KUKA KRL program: MyProgram_325().src

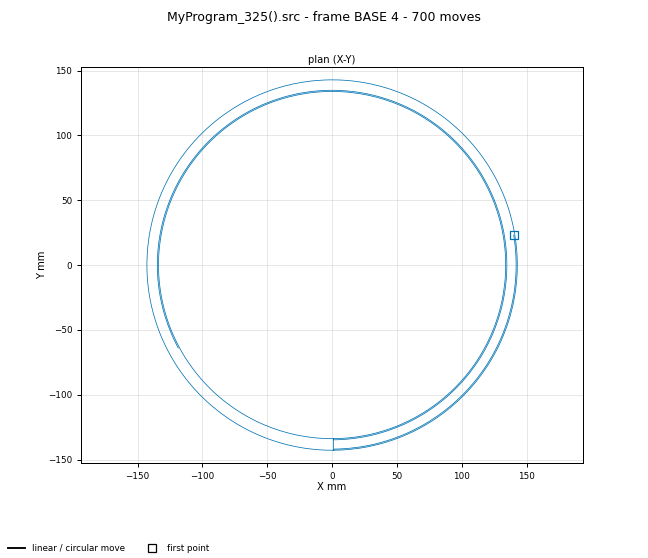
[picture p0: tool path of MyProgram_325().src in frame BASE 4, 700 of 700 moves have a stored position in this frame; points joined in program order, loops and branches not executed]
&ACCESS RVP
&REL 1
&PARAM TEMPLATE = C:\KRC\Roboter\Template\vorgabe
&PARAM EDITMASK = *
DEF MyProgram_325()
; ---- Setting reference (Base) ----
$BASE = BASE_DATA[4]

; --------------------------
; ---- Setting tool (TCP) ----
$TOOL = TOOL_DATA[3]
; --------------------------

$VEL.CP = VEL_APROX_PRINT
Startdeposition()
$VEL.CP = VEL_PRINT
LIN {X 140.0239,Y 23.1296,Z 186,A 12.0919,B 2.8176,C 0.151,E1 2.9796,E2 441.4453} C_DIS
LIN {X 140.5931,Y 19.3826,Z 186,A 10.5222,B 2.8173,C 0.1557,E1 2.9802,E2 443.0211} C_DIS
LIN {X 141.1323,Y 14.9454,Z 186,A 8.8982,B 2.8172,C 0.159,E1 2.9807,E2 444.6224} C_DIS
LIN {X 141.4603,Y 11.4409,Z 186,A 7.6232,B 2.817,C 0.1616,E1 2.981,E2 445.879} C_DIS
LIN {X 141.6829,Y 8.2377,Z 186,A 6.364,B 2.8168,C 0.1649,E1 2.9812,E2 447.1341} C_DIS
LIN {X 141.8322,Y 5.0531,Z 186,A 4.9978,B 2.8166,C 0.1693,E1 2.9814,E2 448.5115} C_DIS
LIN {X 141.9221,Y 0.5024,Z 186,A 3.3333,B 2.8163,C 0.1728,E1 2.9814,E2 450.1543} C_DIS
LIN {X 141.8677,Y -3.9052,Z 186,A 1.6352,B 2.8161,C 0.177,E1 2.9814,E2 451.8427} C_DIS
LIN {X 141.6818,Y -8.2557,Z 186,A -0.0832,B 2.8158,C 0.1816,E1 2.9811,E2 453.557} C_DIS
LIN {X 141.416,Y -11.9653,Z 186,A -1.4595,B 2.8156,C 0.1846,E1 2.9808,E2 454.9177} C_DIS
LIN {X 140.9886,Y -16.2533,Z 186,A -3.1899,B 2.8153,C 0.1894,E1 2.9803,E2 456.648} C_DIS
LIN {X 140.4744,Y -20.2136,Z 186,A -4.647,B 2.8151,C 0.1924,E1 2.9798,E2 458.0855} C_DIS
LIN {X 139.8412,Y -24.2216,Z 186,A -6.1665,B 2.8148,C 0.1958,E1 2.9791,E2 459.5903} C_DIS
LIN {X 139.1946,Y -27.692,Z 186,A -7.6942,B 2.8145,C 0.2007,E1 2.9783,E2 461.1327} C_DIS
LIN {X 138.4456,Y -31.2179,Z 186,A -8.97,B 2.8143,C 0.203,E1 2.9775,E2 462.3856} C_DIS
LIN {X 137.6289,Y -34.6403,Z 186,A -10.6237,B 2.8139,C 0.2092,E1 2.9764,E2 464.0716} C_DIS
LIN {X 136.6827,Y -38.2022,Z 186,A -11.6255,B 2.8139,C 0.2085,E1 2.9757,E2 465.0091} C_DIS
LIN {X 135.7817,Y -41.2912,Z 186,A -13.193,B 2.8135,C 0.2146,E1 2.9744,E2 466.6138} C_DIS
LIN {X 134.8055,Y -44.3763,Z 186,A -14.0659,B 2.8135,C 0.214,E1 2.9737,E2 467.4294} C_DIS
LIN {X 132.8291,Y -49.9801,Z 186,A -16.5006,B 2.813,C 0.2208,E1 2.9714,E2 469.8708} C_DIS
LIN {X 131.2867,Y -53.9078,Z 186,A -18.1056,B 2.8127,C 0.2243,E1 2.9697,E2 471.4639} C_DIS
LIN {X 129.9256,Y -57.1105,Z 186,A -19.7166,B 2.8123,C 0.23,E1 2.9679,E2 473.1038} C_DIS
LIN {X 127.8853,Y -61.5388,Z 186,A -21.3367,B 2.8121,C 0.2317,E1 2.9661,E2 474.6783} C_DIS
LIN {X 126.3115,Y -64.7073,Z 186,A -22.6948,B 2.8119,C 0.2347,E1 2.9644,E2 476.0279} C_DIS
LIN {X 123.5736,Y -69.7979,Z 186,A -24.9173,B 2.8115,C 0.2395,E1 2.9614,E2 478.2372} C_DIS
LIN {X 121.6299,Y -73.1327,Z 186,A -26.5275,B 2.8111,C 0.2439,E1 2.9591,E2 479.8558} C_DIS
LIN {X 119.2262,Y -76.9892,Z 186,A -28.2788,B 2.8108,C 0.2475,E1 2.9565,E2 481.5972} C_DIS
LIN {X 116.8273,Y -80.5827,Z 186,A -29.9461,B 2.8105,C 0.251,E1 2.9539,E2 483.2554} C_DIS
LIN {X 114.225,Y -84.2307,Z 186,A -31.7088,B 2.8101,C 0.2548,E1 2.951,E2 485.0133} C_DIS
LIN {X 112.3154,Y -86.7605,Z 186,A -32.9286,B 2.8099,C 0.2572,E1 2.949,E2 486.2259} C_DIS
LIN {X 109.5218,Y -90.2617,Z 186,A -35.3139,B 2.809,C 0.2665,E1 2.9446,E2 488.6912} C_DIS
LIN {X 105.5037,Y -94.9271,Z 186,A -36.8193,B 2.8094,C 0.263,E1 2.942,E2 490.0649} C_DIS
LIN {X 103.2751,Y -97.3465,Z 186,A -38.3218,B 2.8089,C 0.2675,E1 2.9391,E2 491.5925} C_DIS
LIN {X 100.0952,Y -100.6134,Z 186,A -40.0946,B 2.8086,C 0.2707,E1 2.9357,E2 493.3574} C_DIS
LIN {X 95.9156,Y -104.6055,Z 186,A -42.6088,B 2.808,C 0.277,E1 2.9305,E2 495.8982} C_DIS
LIN {X 93.0795,Y -107.1372,Z 186,A -43.6493,B 2.8082,C 0.2756,E1 2.9284,E2 496.872} C_DIS
LIN {X 90.4094,Y -109.3995,Z 186,A -45.1757,B 2.8078,C 0.2793,E1 2.9251,E2 498.4152} C_DIS
LIN {X 86.8687,Y -112.2316,Z 186,A -47.0306,B 2.8074,C 0.2829,E1 2.921,E2 500.2749} C_DIS
LIN {X 81.8651,Y -115.9319,Z 186,A -49.3362,B 2.8072,C 0.2856,E1 2.9159,E2 502.5539} C_DIS
LIN {X 75.206,Y -120.3587,Z 186,A -52.8874,B 2.8063,C 0.2937,E1 2.9075,E2 506.152} C_DIS
LIN {X 71.5212,Y -122.5846,Z 186,A -54.177,B 2.8064,C 0.2926,E1 2.9045,E2 507.3811} C_DIS
LIN {X 67.7491,Y -124.7085,Z 186,A -55.952,B 2.8061,C 0.2955,E1 2.9001,E2 509.1612} C_DIS
LIN {X 63.7556,Y -126.796,Z 186,A -57.6208,B 2.806,C 0.2968,E1 2.896,E2 510.8105} C_DIS
LIN {X 60.0079,Y -128.6111,Z 186,A -59.6541,B 2.8054,C 0.302,E1 2.8908,E2 512.8937} C_DIS
LIN {X 56.3859,Y -130.2389,Z 186,A -60.8578,B 2.8056,C 0.3007,E1 2.8878,E2 514.0432} C_DIS
LIN {X 53.0905,Y -131.6166,Z 186,A -62.2781,B 2.8054,C 0.3023,E1 2.8842,E2 515.4615} C_DIS
LIN {X 49.9057,Y -132.857,Z 186,A -63.6338,B 2.8053,C 0.3037,E1 2.8806,E2 516.8148} C_DIS
LIN {X 46.6516,Y -134.0344,Z 186,A -65.008,B 2.8051,C 0.3051,E1 2.877,E2 518.1868} C_DIS
LIN {X 42.9116,Y -135.2784,Z 186,A -66.5367,B 2.805,C 0.3062,E1 2.873,E2 519.7079} C_DIS
LIN {X 39.1524,Y -136.4157,Z 186,A -68.0675,B 2.8049,C 0.3073,E1 2.8689,E2 521.2321} C_DIS
LIN {X 36.016,Y -137.2762,Z 186,A -69.4137,B 2.8047,C 0.3087,E1 2.8652,E2 522.5837} C_DIS
LIN {X 32.2587,Y -138.2079,Z 186,A -70.9248,B 2.8047,C 0.3096,E1 2.8611,E2 524.0887} C_DIS
LIN {X 28.5439,Y -139.0213,Z 186,A -72.4888,B 2.8045,C 0.311,E1 2.8568,E2 525.6576} C_DIS
LIN {X 24.7032,Y -139.755,Z 186,A -74.0205,B 2.8044,C 0.3117,E1 2.8526,E2 527.1836} C_DIS
LIN {X 20.1406,Y -140.4848,Z 186,A -75.8828,B 2.8043,C 0.3128,E1 2.8475,E2 529.0465} C_DIS
LIN {X 16.2985,Y -140.9832,Z 186,A -77.3486,B 2.8043,C 0.3129,E1 2.8435,E2 530.4995} C_DIS
LIN {X 13.3998,Y -141.2874,Z 186,A -78.5068,B 2.8042,C 0.3133,E1 2.8402,E2 531.6558} C_DIS
LIN {X 9.8982,Y -141.5764,Z 186,A -80.0763,B 2.804,C 0.315,E1 2.8358,E2 533.2471} C_DIS
LIN {X 5.6109,Y -141.8104,Z 186,A -81.6951,B 2.804,C 0.3147,E1 2.8313,E2 534.8508} C_DIS
LIN {X 1.7593,Y -141.9118,Z 186,A -83.195,B 2.804,C 0.3147,E1 2.8271,E2 536.3438} C_DIS
LIN {X 1.7593,Y -141.9118,Z 186,A -83.195,B 2.804,C 0.3147,E1 2.8271,E2 536.3438} C_DIS
Enddeposition()
LIN {X 1.0264,Y -142.8167,Z 186,A -83.224,B 2.8043,C 0.3144,E1 2.8273,E2 536.3658} C_DIS
Startdeposition()
$VEL.CP = VEL_PRINT
LIN {X 3.5033,Y -142.779,Z 186,A -81.8807,B 2.8046,C 0.3116,E1 2.8312,E2 534.9727} C_DIS
LIN {X 7.0229,Y -142.6485,Z 186,A -80.4898,B 2.8046,C 0.3114,E1 2.835,E2 533.5842} C_DIS
LIN {X 10.5163,Y -142.4335,Z 186,A -79.1018,B 2.8046,C 0.311,E1 2.8389,E2 532.1978} C_DIS
LIN {X 14.0027,Y -142.1335,Z 186,A -77.5929,B 2.8048,C 0.3096,E1 2.8431,E2 530.6732} C_DIS
LIN {X 18.5625,Y -141.6097,Z 186,A -75.8806,B 2.8048,C 0.3096,E1 2.8479,E2 528.9781} C_DIS
LIN {X 21.6541,Y -141.1701,Z 186,A -74.6376,B 2.8048,C 0.3089,E1 2.8513,E2 527.7358} C_DIS
LIN {X 25.1063,Y -140.597,Z 186,A -73.4449,B 2.8048,C 0.3096,E1 2.8545,E2 526.5721} C_DIS
LIN {X 27.8712,Y -140.0764,Z 186,A -72.1321,B 2.805,C 0.3074,E1 2.8582,E2 525.2327} C_DIS
LIN {X 31.4383,Y -139.3183,Z 186,A -70.7315,B 2.8051,C 0.3068,E1 2.862,E2 523.84} C_DIS
LIN {X 34.693,Y -138.5439,Z 186,A -69.3702,B 2.8052,C 0.3055,E1 2.8657,E2 522.4751} C_DIS
LIN {X 38.0738,Y -137.653,Z 186,A -67.9909,B 2.8054,C 0.3044,E1 2.8694,E2 521.0983} C_DIS
LIN {X 42.1178,Y -136.4698,Z 186,A -66.3095,B 2.8055,C 0.3028,E1 2.8739,E2 519.4171} C_DIS
LIN {X 45.8228,Y -135.2723,Z 186,A -64.6461,B 2.8058,C 0.3004,E1 2.8784,E2 517.7384} C_DIS
LIN {X 50.4141,Y -133.6275,Z 186,A -62.7765,B 2.8059,C 0.2989,E1 2.8832,E2 515.8797} C_DIS
LIN {X 54.6585,Y -131.9484,Z 186,A -60.9566,B 2.8062,C 0.2968,E1 2.888,E2 514.0601} C_DIS
LIN {X 59.0093,Y -130.0624,Z 186,A -59.1146,B 2.8064,C 0.2948,E1 2.8926,E2 512.2253} C_DIS
LIN {X 62.6453,Y -128.3498,Z 186,A -57.5736,B 2.8065,C 0.2932,E1 2.8965,E2 510.6933} C_DIS
LIN {X 66.0822,Y -126.6136,Z 186,A -56.1913,B 2.8066,C 0.2924,E1 2.8999,E2 509.3327} C_DIS
LIN {X 69.6422,Y -124.6934,Z 186,A -54.4842,B 2.807,C 0.2893,E1 2.9041,E2 507.6126} C_DIS
LIN {X 73.4813,Y -122.4704,Z 186,A -52.7308,B 2.8072,C 0.2867,E1 2.9083,E2 505.8616} C_DIS
LIN {X 77.1881,Y -120.1681,Z 186,A -51.046,B 2.8075,C 0.2844,E1 2.9123,E2 504.1847} C_DIS
LIN {X 81.086,Y -117.5734,Z 186,A -49.2039,B 2.8077,C 0.2816,E1 2.9165,E2 502.3464} C_DIS
LIN {X 84.8308,Y -114.9007,Z 186,A -47.4602,B 2.808,C 0.2792,E1 2.9204,E2 500.6156} C_DIS
LIN {X 88.3073,Y -112.2504,Z 186,A -45.7728,B 2.8082,C 0.2766,E1 2.9242,E2 498.9362} C_DIS
LIN {X 91.5521,Y -109.6204,Z 186,A -44.1041,B 2.8085,C 0.2735,E1 2.9278,E2 497.2671} C_DIS
LIN {X 94.6507,Y -106.956,Z 186,A -42.5663,B 2.8088,C 0.2712,E1 2.931,E2 495.7422} C_DIS
LIN {X 97.8786,Y -104.0102,Z 186,A -40.837,B 2.8091,C 0.2679,E1 2.9345,E2 494.0149} C_DIS
LIN {X 101.0081,Y -100.9747,Z 186,A -39.1673,B 2.8094,C 0.265,E1 2.9378,E2 492.355} C_DIS
LIN {X 104.0404,Y -97.8466,Z 186,A -37.4658,B 2.8097,C 0.2617,E1 2.9411,E2 490.6586} C_DIS
LIN {X 106.975,Y -94.6291,Z 186,A -35.7918,B 2.8099,C 0.2586,E1 2.9442,E2 488.9933} C_DIS
LIN {X 109.8164,Y -91.3168,Z 186,A -34.0851,B 2.8103,C 0.2551,E1 2.9473,E2 487.2914} C_DIS
LIN {X 112.5897,Y -87.8754,Z 186,A -32.4077,B 2.8105,C 0.252,E1 2.9501,E2 485.6259} C_DIS
LIN {X 115.2422,Y -84.3659,Z 186,A -30.6981,B 2.8109,C 0.2484,E1 2.953,E2 483.9226} C_DIS
LIN {X 117.9636,Y -80.5173,Z 186,A -28.8724,B 2.8112,C 0.2445,E1 2.9559,E2 482.1045} C_DIS
LIN {X 120.4817,Y -76.6982,Z 186,A -27.1511,B 2.8115,C 0.2412,E1 2.9585,E2 480.3975} C_DIS
LIN {X 122.775,Y -72.9702,Z 186,A -25.4865,B 2.8118,C 0.2377,E1 2.9609,E2 478.7442} C_DIS
LIN {X 124.8768,Y -69.3119,Z 186,A -23.8277,B 2.8121,C 0.2338,E1 2.9631,E2 477.0887} C_DIS
LIN {X 127.0236,Y -65.2921,Z 186,A -22.0854,B 2.8124,C 0.23,E1 2.9654,E2 475.3568} C_DIS
LIN {X 128.729,Y -61.8603,Z 186,A -20.6952,B 2.8126,C 0.2275,E1 2.9671,E2 473.9858} C_DIS
LIN {X 130.2185,Y -58.6604,Z 186,A -19.3,B 2.8129,C 0.224,E1 2.9687,E2 472.5923} C_DIS
LIN {X 131.9514,Y -54.6512,Z 186,A -17.6611,B 2.8132,C 0.2205,E1 2.9705,E2 470.9678} C_DIS
LIN {X 133.326,Y -51.2081,Z 186,A -16.2498,B 2.8134,C 0.2173,E1 2.9719,E2 469.5658} C_DIS
LIN {X 134.4941,Y -48.0549,Z 186,A -14.8672,B 2.8137,C 0.2134,E1 2.9732,E2 468.1775} C_DIS
LIN {X 135.9524,Y -43.7587,Z 186,A -13.1073,B 2.8141,C 0.2091,E1 2.9747,E2 466.4245} C_DIS
LIN {X 137.3872,Y -39.0244,Z 186,A -11.2827,B 2.8143,C 0.2052,E1 2.9762,E2 464.6204} C_DIS
LIN {X 138.3747,Y -35.3598,Z 186,A -9.9715,B 2.8145,C 0.2031,E1 2.9771,E2 463.337} C_DIS
LIN {X 139.1148,Y -32.3294,Z 186,A -8.631,B 2.8148,C 0.1988,E1 2.9779,E2 461.9834} C_DIS
LIN {X 139.8672,Y -28.8997,Z 186,A -7.3337,B 2.815,C 0.196,E1 2.9787,E2 460.7003} C_DIS
LIN {X 140.5352,Y -25.4517,Z 186,A -6.1887,B 2.815,C 0.1947,E1 2.9793,E2 459.5903} C_DIS
LIN {X 141.0093,Y -22.6915,Z 186,A -4.9172,B 2.8154,C 0.1901,E1 2.9799,E2 458.2979} C_DIS
LIN {X 141.5249,Y -19.2091,Z 186,A -3.5684,B 2.8156,C 0.1868,E1 2.9804,E2 456.9567} C_DIS
LIN {X 141.9526,Y -15.7335,Z 186,A -2.2335,B 2.8158,C 0.1835,E1 2.9808,E2 455.6303} C_DIS
LIN {X 142.295,Y -12.2497,Z 186,A -0.9002,B 2.816,C 0.1803,E1 2.9811,E2 454.3057} C_DIS
LIN {X 142.5946,Y -8.0731,Z 186,A 0.7864,B 2.8164,C 0.1755,E1 2.9814,E2 452.6171} C_DIS
LIN {X 142.7493,Y -4.5745,Z 186,A 2.1457,B 2.8166,C 0.172,E1 2.9816,E2 451.263} C_DIS
LIN {X 142.8238,Y -0.2041,Z 186,A 3.7721,B 2.8168,C 0.1683,E1 2.9816,E2 449.6528} C_DIS
LIN {X 142.7789,Y 3.5074,Z 186,A 5.1333,B 2.817,C 0.1654,E1 2.9816,E2 448.3079} C_DIS
LIN {X 142.6494,Y 7.0055,Z 186,A 6.4619,B 2.8172,C 0.1621,E1 2.9814,E2 446.9886} C_DIS
LIN {X 142.4132,Y 10.7947,Z 186,A 7.9498,B 2.8174,C 0.1582,E1 2.9811,E2 445.5045} C_DIS
LIN {X 142.0648,Y 14.6902,Z 186,A 9.4152,B 2.8176,C 0.1548,E1 2.9807,E2 444.0523} C_DIS
LIN {X 141.7256,Y 17.6716,Z 186,A 10.5334,B 2.8177,C 0.1523,E1 2.9803,E2 442.9449} C_DIS
LIN {X 141.2773,Y 20.9561,Z 186,A 11.8082,B 2.8179,C 0.1491,E1 2.9798,E2 441.6766} C_DIS
LIN {X 140.7141,Y 24.452,Z 186,A 13.1794,B 2.8181,C 0.1457,E1 2.9792,E2 440.3113} C_DIS
LIN {X 140.0725,Y 27.8908,Z 186,A 14.5133,B 2.8182,C 0.1424,E1 2.9785,E2 438.9859} C_DIS
LIN {X 139.348,Y 31.3081,Z 186,A 15.9331,B 2.8184,C 0.1384,E1 2.9777,E2 437.5628} C_DIS
LIN {X 138.3727,Y 35.3675,Z 186,A 17.3068,B 2.8184,C 0.1367,E1 2.9768,E2 436.2285} C_DIS
LIN {X 137.6519,Y 38.0778,Z 186,A 18.5141,B 2.8187,C 0.1329,E1 2.9759,E2 435.0097} C_DIS
LIN {X 136.47,Y 42.1169,Z 186,A 20.1242,B 2.8189,C 0.129,E1 2.9746,E2 433.4092} C_DIS
LIN {X 135.2768,Y 45.8093,Z 186,A 21.741,B 2.8191,C 0.1243,E1 2.9732,E2 431.7837} C_DIS
LIN {X 133.6282,Y 50.4121,Z 186,A 23.4841,B 2.8192,C 0.1212,E1 2.9715,E2 430.0688} C_DIS
LIN {X 132.3523,Y 53.6724,Z 186,A 24.8259,B 2.8193,C 0.1181,E1 2.9701,E2 428.7346} C_DIS
LIN {X 130.9969,Y 56.9002,Z 186,A 26.2201,B 2.8195,C 0.1145,E1 2.9686,E2 427.3412} C_DIS
LIN {X 129.1131,Y 61.0562,Z 186,A 27.9112,B 2.8196,C 0.1111,E1 2.9666,E2 425.6679} C_DIS
LIN {X 127.4228,Y 64.5079,Z 186,A 29.3877,B 2.8198,C 0.1078,E1 2.9648,E2 424.1994} C_DIS
LIN {X 125.6278,Y 67.9422,Z 186,A 30.9114,B 2.8198,C 0.1042,E1 2.9628,E2 422.6793} C_DIS
LIN {X 123.6588,Y 71.4622,Z 186,A 32.5098,B 2.82,C 0.1003,E1 2.9606,E2 421.083} C_DIS
LIN {X 121.3121,Y 75.3771,Z 186,A 34.2394,B 2.8202,C 0.0968,E1 2.9581,E2 419.3661} C_DIS
LIN {X 119.2399,Y 78.6141,Z 186,A 35.7423,B 2.8202,C 0.0935,E1 2.9558,E2 417.868} C_DIS
LIN {X 116.5772,Y 82.5114,Z 186,A 37.5713,B 2.8204,C 0.0896,E1 2.9529,E2 416.0469} C_DIS
LIN {X 113.8111,Y 86.287,Z 186,A 39.319,B 2.8204,C 0.0865,E1 2.95,E2 414.3158} C_DIS
LIN {X 111.2859,Y 89.5199,Z 186,A 40.952,B 2.8206,C 0.0829,E1 2.9472,E2 412.684} C_DIS
LIN {X 108.4932,Y 92.8855,Z 186,A 42.6555,B 2.8206,C 0.0795,E1 2.9441,E2 410.9868} C_DIS
LIN {X 105.598,Y 96.1636,Z 186,A 44.336,B 2.8208,C 0.0763,E1 2.941,E2 409.3158} C_DIS
LIN {X 102.4606,Y 99.4997,Z 186,A 46.0579,B 2.8208,C 0.0735,E1 2.9377,E2 407.6085} C_DIS
LIN {X 99.4987,Y 102.4615,Z 186,A 47.7266,B 2.8209,C 0.0702,E1 2.9344,E2 405.9412} C_DIS
LIN {X 96.1622,Y 105.5993,Z 186,A 49.4716,B 2.821,C 0.0673,E1 2.9308,E2 404.2079} C_DIS
LIN {X 92.8848,Y 108.4938,Z 186,A 51.1713,B 2.821,C 0.0644,E1 2.9273,E2 402.5152} C_DIS
LIN {X 89.5199,Y 111.2858,Z 186,A 52.8489,B 2.8211,C 0.0618,E1 2.9237,E2 400.8473} C_DIS
LIN {X 86.2062,Y 113.8721,Z 186,A 54.5287,B 2.8211,C 0.0588,E1 2.9199,E2 399.1683} C_DIS
LIN {X 82.5098,Y 116.5783,Z 186,A 56.329,B 2.8213,C 0.056,E1 2.9159,E2 397.3729} C_DIS
LIN {X 78.6138,Y 119.2401,Z 186,A 58.1375,B 2.8213,C 0.0535,E1 2.9117,E2 395.5753} C_DIS
LIN {X 74.9259,Y 121.5916,Z 186,A 59.8568,B 2.8213,C 0.051,E1 2.9076,E2 393.8607} C_DIS
LIN {X 71.167,Y 123.8297,Z 186,A 61.6008,B 2.8213,C 0.0484,E1 2.9034,E2 392.1181} C_DIS
LIN {X 67.3103,Y 125.9673,Z 186,A 63.3155,B 2.8214,C 0.0463,E1 2.8992,E2 390.4105} C_DIS
LIN {X 63.4165,Y 127.9693,Z 186,A 64.9047,B 2.8214,C 0.0452,E1 2.8953,E2 388.843} C_DIS
LIN {X 60.2641,Y 129.484,Z 186,A 66.2752,B 2.8214,C 0.0436,E1 2.8919,E2 387.4767} C_DIS
LIN {X 56.9023,Y 130.996,Z 186,A 67.8358,B 2.8215,C 0.0412,E1 2.8878,E2 385.9059} C_DIS
LIN {X 53.0242,Y 132.6135,Z 186,A 69.3772,B 2.8215,C 0.0403,E1 2.8839,E2 384.3833} C_DIS
LIN {X 49.756,Y 133.874,Z 186,A 70.7622,B 2.8215,C 0.0389,E1 2.8803,E2 383.0011} C_DIS
LIN {X 45.767,Y 135.2909,Z 186,A 72.5173,B 2.8215,C 0.0367,E1 2.8756,E2 381.2391} C_DIS
LIN {X 41.4185,Y 136.6838,Z 186,A 74.3145,B 2.8215,C 0.0352,E1 2.8708,E2 379.4467} C_DIS
LIN {X 37.2433,Y 137.8802,Z 186,A 75.9865,B 2.8216,C 0.0341,E1 2.8664,E2 377.7841} C_DIS
LIN {X 34.0209,Y 138.7109,Z 186,A 77.2564,B 2.8216,C 0.0335,E1 2.8629,E2 376.5229} C_DIS
LIN {X 30.6107,Y 139.5028,Z 186,A 78.6422,B 2.8216,C 0.0326,E1 2.8592,E2 375.1398} C_DIS
LIN {X 26.8278,Y 140.2787,Z 186,A 80.1703,B 2.8216,C 0.0317,E1 2.855,E2 373.6148} C_DIS
LIN {X 23.3684,Y 140.8963,Z 186,A 81.5622,B 2.8216,C 0.031,E1 2.8512,E2 372.2257} C_DIS
LIN {X 20.2637,Y 141.3762,Z 186,A 82.8111,B 2.8216,C 0.0304,E1 2.8477,E2 370.9786} C_DIS
LIN {X 16.4181,Y 141.8752,Z 186,A 84.3496,B 2.8216,C 0.0297,E1 2.8434,E2 369.4428} C_DIS
LIN {X 12.2492,Y 142.2951,Z 186,A 86.0263,B 2.8216,C 0.0291,E1 2.8388,E2 367.7672} C_DIS
LIN {X 8.0728,Y 142.5946,Z 186,A 87.7919,B 2.8216,C 0.028,E1 2.8338,E2 365.9914} C_DIS
LIN {X 4.5608,Y 142.7496,Z 186,A 89.1132,B 2.8216,C 0.0282,E1 2.8302,E2 364.6821} C_DIS
LIN {X 1.0584,Y 142.8176,Z 186,A 90.2879,B 2.8216,C 0.0295,E1 2.827,E2 363.5372} C_DIS
LIN {X -1.7572,Y 142.8118,Z 186,A 91.6431,B 2.8216,C 0.0279,E1 2.8231,E2 362.1539} C_DIS
LIN {X -5.2564,Y 142.7248,Z 186,A 93.0413,B 2.8216,C 0.0279,E1 2.8192,E2 360.757} C_DIS
LIN {X -8.7802,Y 142.551,Z 186,A 94.4428,B 2.8216,C 0.0279,E1 2.8153,E2 359.3579} C_DIS
LIN {X -12.269,Y 142.2934,Z 186,A 95.8428,B 2.8216,C 0.0281,E1 2.8114,E2 357.9589} C_DIS
LIN {X -16.4294,Y 141.8738,Z 186,A 97.6204,B 2.8216,C 0.0278,E1 2.8064,E2 356.1695} C_DIS
LIN {X -20.2992,Y 141.3712,Z 186,A 99.0382,B 2.8216,C 0.0291,E1 2.8025,E2 354.7712} C_DIS
LIN {X -23.4035,Y 140.8905,Z 186,A 100.3733,B 2.8216,C 0.0291,E1 2.7988,E2 353.4272} C_DIS
LIN {X -26.1764,Y 140.4032,Z 186,A 101.5161,B 2.8216,C 0.0294,E1 2.7957,E2 352.2834} C_DIS
LIN {X -29.6014,Y 139.7207,Z 186,A 102.9252,B 2.8216,C 0.0299,E1 2.7918,E2 350.874} C_DIS
LIN {X -33.004,Y 138.956,Z 186,A 104.335,B 2.8216,C 0.0306,E1 2.788,E2 349.4636} C_DIS
LIN {X -36.3853,Y 138.109,Z 186,A 105.7469,B 2.8216,C 0.0313,E1 2.7841,E2 348.0508} C_DIS
LIN {X -39.786,Y 137.1678,Z 186,A 107.3035,B 2.8216,C 0.0314,E1 2.7799,E2 346.477} C_DIS
LIN {X -43.7901,Y 135.9424,Z 186,A 108.9142,B 2.8216,C 0.033,E1 2.7756,E2 344.8761} C_DIS
LIN {X -48.1524,Y 134.459,Z 186,A 110.8756,B 2.8216,C 0.0339,E1 2.7704,E2 342.9014} C_DIS
LIN {X -52.4959,Y 132.8254,Z 186,A 112.7939,B 2.8216,C 0.0353,E1 2.7654,E2 340.9771} C_DIS
LIN {X -56.9061,Y 130.9943,Z 186,A 114.6555,B 2.8216,C 0.0374,E1 2.7606,E2 339.1236} C_DIS
LIN {X -61.0535,Y 129.1144,Z 186,A 116.4541,B 2.8216,C 0.0395,E1 2.7561,E2 337.3298} C_DIS
LIN {X -64.2233,Y 127.5677,Z 186,A 117.9933,B 2.8216,C 0.0405,E1 2.7522,E2 335.7756} C_DIS
LIN {X -67.6327,Y 125.7941,Z 186,A 119.5665,B 2.8215,C 0.0422,E1 2.7483,E2 334.1994} C_DIS
LIN {X -71.4733,Y 123.6523,Z 186,A 121.3743,B 2.8215,C 0.0443,E1 2.7439,E2 332.3873} C_DIS
LIN {X -75.3817,Y 121.3092,Z 186,A 123.2221,B 2.8215,C 0.0467,E1 2.7395,E2 330.5382} C_DIS
LIN {X -79.056,Y 118.9477,Z 186,A 125.0876,B 2.8214,C 0.0487,E1 2.7351,E2 328.6594} C_DIS
LIN {X -82.9652,Y 116.2545,Z 186,A 127.0099,B 2.8214,C 0.0515,E1 2.7307,E2 326.7361} C_DIS
LIN {X -86.4856,Y 113.6604,Z 186,A 128.8327,B 2.8213,C 0.054,E1 2.7266,E2 324.9059} C_DIS
LIN {X -89.9248,Y 110.9593,Z 186,A 130.5978,B 2.8213,C 0.0569,E1 2.7227,E2 323.1406} C_DIS
LIN {X -93.3335,Y 108.1074,Z 186,A 132.4565,B 2.8212,C 0.0597,E1 2.7188,E2 321.2735} C_DIS
LIN {X -96.5673,Y 105.2288,Z 186,A 134.2343,B 2.8212,C 0.0626,E1 2.7151,E2 319.4917} C_DIS
LIN {X -99.744,Y 102.2232,Z 186,A 136.0961,B 2.8211,C 0.0655,E1 2.7113,E2 317.6173} C_DIS
LIN {X -102.8271,Y 99.1212,Z 186,A 137.912,B 2.821,C 0.0686,E1 2.7077,E2 315.7948} C_DIS
LIN {X -106.064,Y 95.6501,Z 186,A 139.8953,B 2.8209,C 0.0722,E1 2.704,E2 313.8027} C_DIS
LIN {X -109.0631,Y 92.2155,Z 186,A 141.7503,B 2.8208,C 0.0759,E1 2.7006,E2 311.9458} C_DIS
LIN {X -111.8416,Y 88.8246,Z 186,A 143.5632,B 2.8207,C 0.0794,E1 2.6974,E2 310.1272} C_DIS
LIN {X -114.4675,Y 85.4139,Z 186,A 145.394,B 2.8206,C 0.0828,E1 2.6943,E2 308.2843} C_DIS
LIN {X -117.0379,Y 81.857,Z 186,A 147.2351,B 2.8205,C 0.0864,E1 2.6913,E2 306.434} C_DIS
LIN {X -119.5352,Y 78.1656,Z 186,A 149.0884,B 2.8204,C 0.0903,E1 2.6884,E2 304.5736} C_DIS
LIN {X -121.9301,Y 74.374,Z 186,A 150.931,B 2.8202,C 0.0944,E1 2.6857,E2 302.7267} C_DIS
LIN {X -124.0942,Y 70.7032,Z 186,A 152.7303,B 2.8202,C 0.0982,E1 2.6832,E2 300.917} C_DIS
LIN {X -126.1987,Y 66.8723,Z 186,A 154.6009,B 2.82,C 0.102,E1 2.6807,E2 299.0324} C_DIS
LIN {X -127.9623,Y 63.4307,Z 186,A 156.1391,B 2.8198,C 0.1059,E1 2.6787,E2 297.497} C_DIS
LIN {X -129.4885,Y 60.2545,Z 186,A 157.6142,B 2.8197,C 0.1093,E1 2.677,E2 296.0151} C_DIS
LIN {X -130.9998,Y 56.8935,Z 186,A 159.2865,B 2.8196,C 0.1124,E1 2.675,E2 294.3184} C_DIS
LIN {X -132.6119,Y 53.0284,Z 186,A 160.9536,B 2.8194,C 0.1168,E1 2.6733,E2 292.6543} C_DIS
LIN {X -133.871,Y 49.764,Z 186,A 162.4043,B 2.8192,C 0.1203,E1 2.6719,E2 291.1984} C_DIS
LIN {X -135.2743,Y 45.8167,Z 186,A 164.2752,B 2.8191,C 0.1241,E1 2.6701,E2 289.3038} C_DIS
LIN {X -136.4698,Y 42.1178,Z 186,A 165.9356,B 2.8189,C 0.1279,E1 2.6687,E2 287.6312} C_DIS
LIN {X -137.6484,Y 38.0904,Z 186,A 167.5752,B 2.8187,C 0.1326,E1 2.6675,E2 285.9987} C_DIS
LIN {X -138.7071,Y 34.0368,Z 186,A 169.3978,B 2.8185,C 0.1367,E1 2.6662,E2 284.1585} C_DIS
LIN {X -139.5096,Y 30.5796,Z 186,A 170.8456,B 2.8183,C 0.1405,E1 2.6653,E2 282.7087} C_DIS
LIN {X -140.2136,Y 27.168,Z 186,A 172.1198,B 2.8181,C 0.1448,E1 2.6646,E2 281.4517} C_DIS
LIN {X -140.7198,Y 24.4201,Z 186,A 173.4883,B 2.818,C 0.1471,E1 2.6639,E2 280.0512} C_DIS
LIN {X -141.2808,Y 20.9316,Z 186,A 174.9994,B 2.8178,C 0.1507,E1 2.6633,E2 278.5287} C_DIS
LIN {X -141.7505,Y 17.4633,Z 186,A 176.4752,B 2.8176,C 0.1544,E1 2.6628,E2 277.0443} C_DIS
LIN {X -142.1349,Y 13.9879,Z 186,A 177.9486,B 2.8174,C 0.158,E1 2.6623,E2 275.5625} C_DIS
LIN {X -142.4342,Y 10.5065,Z 186,A 179.5099,B 2.8172,C 0.1614,E1 2.662,E2 273.9808} C_DIS
LIN {X -142.6987,Y 5.9266,Z 186,A -178.7431,B 2.8169,C 0.1669,E1 2.6617,E2 272.2475} C_DIS
LIN {X -142.7944,Y 2.8057,Z 186,A -177.4888,B 2.8167,C 0.1704,E1 2.6617,E2 270.9939} C_DIS
LIN {X -142.8222,Y -0.4607,Z 186,A -175.8287,B 2.8165,C 0.1729,E1 2.6617,E2 269.2878} C_DIS
LIN {X -142.7494,Y -4.5692,Z 186,A -174.0501,B 2.8163,C 0.1771,E1 2.6617,E2 267.4928} C_DIS
LIN {X -142.5518,Y -8.768,Z 186,A -172.4295,B 2.8159,C 0.1821,E1 2.662,E2 265.882} C_DIS
LIN {X -142.2919,Y -12.2873,Z 186,A -170.9451,B 2.8157,C 0.1858,E1 2.6623,E2 264.3893} C_DIS
LIN {X -141.8731,Y -16.4351,Z 186,A -169.0846,B 2.8154,C 0.1898,E1 2.6629,E2 262.5044} C_DIS
LIN {X -141.3397,Y -20.5192,Z 186,A -167.4044,B 2.8151,C 0.1943,E1 2.6636,E2 260.8214} C_DIS
LIN {X -140.7241,Y -24.3964,Z 186,A -165.7692,B 2.8148,C 0.1985,E1 2.6643,E2 259.1789} C_DIS
LIN {X -140.0851,Y -27.8288,Z 186,A -164.1747,B 2.8146,C 0.2016,E1 2.6652,E2 257.5589} C_DIS
LIN {X -139.3525,Y -31.2887,Z 186,A -162.7101,B 2.8143,C 0.2053,E1 2.6661,E2 256.0888} C_DIS
LIN {X -138.3712,Y -35.3734,Z 186,A -161.001,B 2.814,C 0.2098,E1 2.6672,E2 254.3773} C_DIS
LIN {X -137.3608,Y -39.1187,Z 186,A -159.2495,B 2.8137,C 0.2133,E1 2.6685,E2 252.6001} C_DIS
LIN {X -135.944,Y -43.7851,Z 186,A -157.313,B 2.8133,C 0.2186,E1 2.6702,E2 250.6672} C_DIS
LIN {X -134.4662,Y -48.1322,Z 186,A -155.2888,B 2.813,C 0.2227,E1 2.672,E2 248.619} C_DIS
LIN {X -133.0005,Y -52.0456,Z 186,A -153.6546,B 2.8127,C 0.2273,E1 2.6737,E2 246.9913} C_DIS
LIN {X -131.6861,Y -55.2865,Z 186,A -152.1833,B 2.8124,C 0.2306,E1 2.6752,E2 245.5113} C_DIS
LIN {X -130.0759,Y -58.9791,Z 186,A -150.3713,B 2.8121,C 0.2339,E1 2.6773,E2 243.6732} C_DIS
LIN {X -128.3509,Y -62.643,Z 186,A -148.7967,B 2.8117,C 0.2382,E1 2.6792,E2 242.106} C_DIS
LIN {X -126.6138,Y -66.0818,Z 186,A -147.2197,B 2.8114,C 0.2418,E1 2.6812,E2 240.5253} C_DIS
LIN {X -124.693,Y -69.6428,Z 186,A -145.4008,B 2.8112,C 0.245,E1 2.6837,E2 238.68} C_DIS
LIN {X -122.5029,Y -73.4267,Z 186,A -143.5366,B 2.8108,C 0.2487,E1 2.6864,E2 236.8013} C_DIS
LIN {X -120.1981,Y -77.1412,Z 186,A -141.8114,B 2.8105,C 0.2529,E1 2.6889,E2 235.0804} C_DIS
LIN {X -117.9639,Y -80.517,Z 186,A -139.988,B 2.8102,C 0.2557,E1 2.6918,E2 233.23} C_DIS
LIN {X -115.4236,Y -84.118,Z 186,A -138.2108,B 2.8099,C 0.2596,E1 2.6947,E2 231.452} C_DIS
LIN {X -112.7949,Y -87.6108,Z 186,A -136.4038,B 2.8095,C 0.2631,E1 2.6978,E2 229.6379} C_DIS
LIN {X -110.0635,Y -91.0184,Z 186,A -134.5215,B 2.8092,C 0.2662,E1 2.7012,E2 227.7379} C_DIS
LIN {X -106.9878,Y -94.6146,Z 186,A -132.6063,B 2.8089,C 0.27,E1 2.7047,E2 225.8208} C_DIS
LIN {X -104.6371,Y -97.2082,Z 186,A -131.1418,B 2.8086,C 0.2725,E1 2.7075,E2 224.3481} C_DIS
LIN {X -101.6105,Y -100.3683,Z 186,A -129.3078,B 2.8083,C 0.2755,E1 2.7111,E2 222.5034} C_DIS
LIN {X -98.4713,Y -103.4495,Z 186,A -127.4637,B 2.8081,C 0.2784,E1 2.7148,E2 220.6485} C_DIS
LIN {X -95.2631,Y -106.4108,Z 186,A -125.6734,B 2.8078,C 0.2813,E1 2.7185,E2 218.8529} C_DIS
LIN {X -91.9499,Y -109.2867,Z 186,A -123.8713,B 2.8075,C 0.2841,E1 2.7224,E2 217.0451} C_DIS
LIN {X -88.5574,Y -112.054,Z 186,A -122.0126,B 2.8072,C 0.2865,E1 2.7264,E2 215.1721} C_DIS
LIN {X -85.0672,Y -114.7257,Z 186,A -120.2562,B 2.807,C 0.2893,E1 2.7304,E2 213.4167} C_DIS
LIN {X -81.5148,Y -117.276,Z 186,A -118.4569,B 2.8067,C 0.2917,E1 2.7345,E2 211.6111} C_DIS
LIN {X -77.8872,Y -119.716,Z 186,A -116.6203,B 2.8065,C 0.2937,E1 2.7388,E2 209.7629} C_DIS
LIN {X -74.1754,Y -122.051,Z 186,A -114.8048,B 2.8063,C 0.2958,E1 2.7431,E2 207.9393} C_DIS
LIN {X -70.2967,Y -124.3255,Z 186,A -112.9721,B 2.8061,C 0.2979,E1 2.7476,E2 206.1024} C_DIS
LIN {X -66.8419,Y -126.2147,Z 186,A -111.4542,B 2.8058,C 0.3001,E1 2.7513,E2 204.5929} C_DIS
LIN {X -63.4222,Y -127.9665,Z 186,A -109.8782,B 2.8057,C 0.3016,E1 2.7552,E2 203.0119} C_DIS
LIN {X -60.2707,Y -129.481,Z 186,A -108.4489,B 2.8055,C 0.3029,E1 2.7589,E2 201.5786} C_DIS
LIN {X -56.5025,Y -131.1688,Z 186,A -106.7252,B 2.8054,C 0.3042,E1 2.7633,E2 199.8452} C_DIS
LIN {X -53.0272,Y -132.6123,Z 186,A -105.2162,B 2.8052,C 0.3055,E1 2.7672,E2 198.336} C_DIS
LIN {X -49.6953,Y -133.8967,Z 186,A -103.77,B 2.8052,C 0.3066,E1 2.771,E2 196.8875} C_DIS
LIN {X -45.7838,Y -135.2853,Z 186,A -101.9837,B 2.8051,C 0.3072,E1 2.7758,E2 195.0838} C_DIS
LIN {X -41.3396,Y -136.7079,Z 186,A -100.1007,B 2.8049,C 0.3083,E1 2.7808,E2 193.1988} C_DIS
LIN {X -37.4166,Y -137.834,Z 186,A -98.4359,B 2.8049,C 0.3091,E1 2.7853,E2 191.5296} C_DIS
LIN {X -34.0263,Y -138.7096,Z 186,A -97.1107,B 2.8047,C 0.3103,E1 2.7889,E2 190.2152} C_DIS
LIN {X -30.1632,Y -139.5994,Z 186,A -95.4357,B 2.8047,C 0.3105,E1 2.7935,E2 188.5277} C_DIS
LIN {X -26.1447,Y -140.4092,Z 186,A -93.8659,B 2.8046,C 0.3116,E1 2.7978,E2 186.968} C_DIS
LIN {X -22.6778,Y -141.0115,Z 186,A -92.4267,B 2.8046,C 0.3118,E1 2.8017,E2 185.5244} C_DIS
LIN {X -19.2134,Y -141.5244,Z 186,A -91.0156,B 2.8046,C 0.312,E1 2.8056,E2 184.1118} C_DIS
LIN {X -15.7381,Y -141.9521,Z 186,A -89.6104,B 2.8045,C 0.3122,E1 2.8096,E2 182.7061} C_DIS
LIN {X -12.2537,Y -142.2947,Z 186,A -88.2086,B 2.8045,C 0.3124,E1 2.8135,E2 181.304} C_DIS
LIN {X -8.0647,Y -142.5951,Z 186,A -86.4303,B 2.8045,C 0.3117,E1 2.8185,E2 179.5118} C_DIS
LIN {X -4.5644,Y -142.7495,Z 186,A -85.1076,B 2.8045,C 0.3122,E1 2.8221,E2 178.2002} C_DIS
LIN {X -1.0623,Y -142.8176,Z 186,A -83.9293,B 2.8043,C 0.3136,E1 2.8253,E2 177.0533} C_DIS
LIN {X 1.0264,Y -142.8167,Z 186,A -83.2235,B 2.8043,C 0.3144,E1 2.8273,E2 176.3657} C_DIS
Enddeposition()
LIN {X 0.9691,Y -133.8678,Z 187,A -82.8691,B 2.3885,C 0.2815,E1 2.4113,E2 175.7764} C_DIS
Startdeposition()
$VEL.CP = VEL_PRINT
LIN {X -2.8245,Y -133.8434,Z 187,A -84.9056,B 2.3882,C 0.2841,E1 2.4055,E2 177.8679} C_DIS
LIN {X -6.581,Y -133.71,Z 187,A -86.3971,B 2.3882,C 0.2836,E1 2.4013,E2 179.3448} C_DIS
LIN {X -10.3502,Y -133.4724,Z 187,A -88.1612,B 2.3882,C 0.2844,E1 2.3963,E2 181.1289} C_DIS
LIN {X -14.2535,Y -133.1108,Z 187,A -89.6968,B 2.3882,C 0.2835,E1 2.3921,E2 182.6467} C_DIS
LIN {X -17.537,Y -132.7181,Z 187,A -91.1608,B 2.3882,C 0.2835,E1 2.388,E2 184.1175} C_DIS
LIN {X -20.7833,Y -132.2489,Z 187,A -92.4949,B 2.3883,C 0.2829,E1 2.3844,E2 185.4431} C_DIS
LIN {X -24.0173,Y -131.7003,Z 187,A -93.9269,B 2.3883,C 0.2827,E1 2.3804,E2 186.8793} C_DIS
LIN {X -27.2365,Y -131.0728,Z 187,A -95.3165,B 2.3884,C 0.2821,E1 2.3766,E2 188.2676} C_DIS
LIN {X -30.4576,Y -130.3624,Z 187,A -96.7667,B 2.3884,C 0.2817,E1 2.3726,E2 189.7232} C_DIS
LIN {X -33.6439,Y -129.577,Z 187,A -98.1873,B 2.3885,C 0.2811,E1 2.3688,E2 191.1464} C_DIS
LIN {X -36.8099,Y -128.7137,Z 187,A -99.6103,B 2.3886,C 0.2804,E1 2.3649,E2 192.5723} C_DIS
LIN {X -39.9537,Y -127.7729,Z 187,A -101.0357,B 2.3886,C 0.2796,E1 2.3611,E2 194.0007} C_DIS
LIN {X -43.0701,Y -126.7564,Z 187,A -102.4627,B 2.3888,C 0.2788,E1 2.3573,E2 195.4312} C_DIS
LIN {X -46.1998,Y -125.6494,Z 187,A -104.0478,B 2.3888,C 0.2784,E1 2.3531,E2 197.0381} C_DIS
LIN {X -49.717,Y -124.2976,Z 187,A -105.5448,B 2.3891,C 0.2766,E1 2.3492,E2 198.5203} C_DIS
LIN {X -52.7489,Y -123.0416,Z 187,A -106.9759,B 2.3891,C 0.2754,E1 2.3455,E2 199.9552} C_DIS
LIN {X -55.7493,Y -121.7118,Z 187,A -108.4087,B 2.3893,C 0.2741,E1 2.3418,E2 201.3918} C_DIS
LIN {X -59.1613,Y -120.0894,Z 187,A -110.1167,B 2.3895,C 0.2728,E1 2.3375,E2 203.112} C_DIS
LIN {X -62.6689,Y -118.2977,Z 187,A -111.7596,B 2.3897,C 0.2708,E1 2.3334,E2 204.7495} C_DIS
LIN {X -66.0061,Y -116.4706,Z 187,A -113.4579,B 2.3899,C 0.2691,E1 2.3293,E2 206.4571} C_DIS
LIN {X -68.8256,Y -114.8269,Z 187,A -114.9061,B 2.3901,C 0.2676,E1 2.3258,E2 207.9121} C_DIS
LIN {X -71.6253,Y -113.1014,Z 187,A -116.4453,B 2.3902,C 0.2662,E1 2.3221,E2 209.4685} C_DIS
LIN {X -75.3231,Y -110.6734,Z 187,A -118.3062,B 2.3905,C 0.2634,E1 2.3178,E2 211.3252} C_DIS
LIN {X -78.0116,Y -108.7947,Z 187,A -119.7524,B 2.3907,C 0.2615,E1 2.3144,E2 212.777} C_DIS
LIN {X -80.6656,Y -106.8415,Z 187,A -121.293,B 2.3909,C 0.2598,E1 2.3109,E2 214.3344} C_DIS
LIN {X -84.1047,Y -104.156,Z 187,A -123.1857,B 2.3912,C 0.2569,E1 2.3068,E2 216.2303} C_DIS
LIN {X -87.0115,Y -101.7409,Z 187,A -124.9462,B 2.3915,C 0.2547,E1 2.303,E2 218.0091} C_DIS
LIN {X -90.3255,Y -98.8104,Z 187,A -126.8446,B 2.3918,C 0.2514,E1 2.299,E2 219.9081} C_DIS
LIN {X -93.3228,Y -95.9843,Z 187,A -128.6579,B 2.3921,C 0.2483,E1 2.2954,E2 221.7277} C_DIS
LIN {X -96.2869,Y -93.0103,Z 187,A -130.5559,B 2.3925,C 0.2453,E1 2.2916,E2 223.6384} C_DIS
LIN {X -99.1977,Y -89.8993,Z 187,A -132.5015,B 2.3928,C 0.2421,E1 2.2879,E2 225.5993} C_DIS
LIN {X -102.0668,Y -86.6281,Z 187,A -134.4495,B 2.3931,C 0.2386,E1 2.2843,E2 227.558} C_DIS
LIN {X -104.8743,Y -83.2074,Z 187,A -136.4215,B 2.3935,C 0.2349,E1 2.2808,E2 229.5396} C_DIS
LIN {X -107.523,Y -79.7554,Z 187,A -138.2797,B 2.3939,C 0.2308,E1 2.2777,E2 231.3968} C_DIS
LIN {X -109.4504,Y -77.0887,Z 187,A -139.7576,B 2.3942,C 0.2279,E1 2.2753,E2 232.8834} C_DIS
LIN {X -111.315,Y -74.371,Z 187,A -141.2341,B 2.3945,C 0.2249,E1 2.273,E2 234.3678} C_DIS
LIN {X -113.3708,Y -71.1984,Z 187,A -143.0744,B 2.3947,C 0.2218,E1 2.2702,E2 236.236} C_DIS
LIN {X -115.2728,Y -68.076,Z 187,A -144.6525,B 2.3951,C 0.2182,E1 2.2679,E2 237.8153} C_DIS
LIN {X -117.0457,Y -64.9798,Z 187,A -146.1882,B 2.3954,C 0.2146,E1 2.2658,E2 239.3515} C_DIS
LIN {X -118.8259,Y -61.663,Z 187,A -147.9,B 2.3957,C 0.2109,E1 2.2635,E2 241.0756} C_DIS
LIN {X -120.0866,Y -59.1668,Z 187,A -149.1557,B 2.396,C 0.2081,E1 2.262,E2 242.3382} C_DIS
LIN {X -121.5067,Y -56.1929,Z 187,A -150.6447,B 2.3963,C 0.2048,E1 2.2602,E2 243.8366} C_DIS
LIN {X -122.8475,Y -53.1981,Z 187,A -152.1284,B 2.3965,C 0.2015,E1 2.2585,E2 245.3297} C_DIS
LIN {X -124.1145,Y -50.1712,Z 187,A -153.6146,B 2.3968,C 0.1981,E1 2.2569,E2 246.8256} C_DIS
LIN {X -125.485,Y -46.6387,Z 187,A -155.333,B 2.3972,C 0.1941,E1 2.2552,E2 248.5555} C_DIS
LIN {X -126.5897,Y -43.5512,Z 187,A -156.8344,B 2.3974,C 0.1906,E1 2.2538,E2 250.0686} C_DIS
LIN {X -127.6415,Y -40.3654,Z 187,A -158.3361,B 2.3977,C 0.187,E1 2.2525,E2 251.578} C_DIS
LIN {X -128.5518,Y -37.3639,Z 187,A -159.7692,B 2.398,C 0.1836,E1 2.2513,E2 253.0217} C_DIS
LIN {X -129.4516,Y -34.1175,Z 187,A -161.2914,B 2.3983,C 0.1799,E1 2.2502,E2 254.5532} C_DIS
LIN {X -130.2496,Y -30.9324,Z 187,A -162.7818,B 2.3985,C 0.1763,E1 2.2492,E2 256.0536} C_DIS
LIN {X -130.9694,Y -27.729,Z 187,A -164.2714,B 2.3988,C 0.1726,E1 2.2483,E2 257.553} C_DIS
LIN {X -131.6104,Y -24.5093,Z 187,A -165.7616,B 2.3991,C 0.169,E1 2.2475,E2 259.0531} C_DIS
LIN {X -132.1744,Y -21.2634,Z 187,A -167.2819,B 2.3993,C 0.1653,E1 2.2468,E2 260.5863} C_DIS
LIN {X -132.5866,Y -18.5093,Z 187,A -168.6286,B 2.3995,C 0.1623,E1 2.2463,E2 261.9515} C_DIS
LIN {X -133.0564,Y -14.7587,Z 187,A -170.2667,B 2.3998,C 0.1579,E1 2.2457,E2 263.5912} C_DIS
LIN {X -133.3783,Y -11.4854,Z 187,A -171.6711,B 2.4001,C 0.1539,E1 2.2454,E2 264.9943} C_DIS
LIN {X -133.6508,Y -7.706,Z 187,A -173.6318,B 2.4003,C 0.1501,E1 2.245,E2 266.9958} C_DIS
LIN {X -133.8184,Y -3.7833,Z 187,A -175.3372,B 2.4006,C 0.1454,E1 2.2448,E2 268.7033} C_DIS
LIN {X -133.8731,Y -0.1052,Z 187,A -176.8928,B 2.4009,C 0.1409,E1 2.2448,E2 270.2557} C_DIS
LIN {X -133.8442,Y 2.7762,Z 187,A -178.3827,B 2.401,C 0.138,E1 2.2448,E2 271.7762} C_DIS
LIN {X -133.7105,Y 6.5705,Z 187,A -179.988,B 2.4013,C 0.1334,E1 2.2451,E2 273.3781} C_DIS
LIN {X -133.4729,Y 10.344,Z 187,A 178.1321,B 2.4015,C 0.1294,E1 2.2454,E2 275.2888} C_DIS
LIN {X -133.1106,Y 14.2549,Z 187,A 176.5048,B 2.4018,C 0.1246,E1 2.2459,E2 276.9084} C_DIS
LIN {X -132.7213,Y 17.5127,Z 187,A 174.9546,B 2.402,C 0.1209,E1 2.2464,E2 278.4754} C_DIS
LIN {X -132.2498,Y 20.7774,Z 187,A 173.517,B 2.4021,C 0.1171,E1 2.247,E2 279.9152} C_DIS
LIN {X -131.701,Y 24.0134,Z 187,A 171.8435,B 2.4023,C 0.1137,E1 2.2479,E2 281.6203} C_DIS
LIN {X -131.069,Y 27.255,Z 187,A 170.4959,B 2.4025,C 0.1097,E1 2.2486,E2 282.959} C_DIS
LIN {X -130.335,Y 30.5776,Z 187,A 168.9765,B 2.4027,C 0.1059,E1 2.2496,E2 284.4851} C_DIS
LIN {X -129.5764,Y 33.6465,Z 187,A 167.538,B 2.4028,C 0.1024,E1 2.2505,E2 285.933} C_DIS
LIN {X -128.708,Y 36.8304,Z 187,A 166.0359,B 2.403,C 0.0987,E1 2.2517,E2 287.4449} C_DIS
LIN {X -127.7705,Y 39.9614,Z 187,A 164.5513,B 2.4031,C 0.0952,E1 2.2529,E2 288.9388} C_DIS
LIN {X -126.7567,Y 43.0692,Z 187,A 163.0602,B 2.4033,C 0.0916,E1 2.2542,E2 290.4399} C_DIS
LIN {X -125.6563,Y 46.1815,Z 187,A 161.4142,B 2.4033,C 0.0884,E1 2.2558,E2 292.1129} C_DIS
LIN {X -124.3019,Y 49.7063,Z 187,A 159.8596,B 2.4035,C 0.0841,E1 2.2574,E2 293.6589} C_DIS
LIN {X -123.0467,Y 52.7373,Z 187,A 158.3751,B 2.4036,C 0.0807,E1 2.259,E2 295.152} C_DIS
LIN {X -121.7181,Y 55.7357,Z 187,A 156.8864,B 2.4038,C 0.0773,E1 2.2607,E2 296.6498} C_DIS
LIN {X -120.3086,Y 58.7169,Z 187,A 155.499,B 2.4038,C 0.0737,E1 2.2624,E2 298.0333} C_DIS
LIN {X -119.0517,Y 61.2251,Z 187,A 154.1209,B 2.4039,C 0.0711,E1 2.2642,E2 299.4317} C_DIS
LIN {X -117.2788,Y 64.559,Z 187,A 152.4281,B 2.4041,C 0.0673,E1 2.2664,E2 301.1324} C_DIS
LIN {X -115.6616,Y 67.4137,Z 187,A 150.9367,B 2.4041,C 0.0642,E1 2.2685,E2 302.6332} C_DIS
LIN {X -113.9755,Y 70.2261,Z 187,A 149.4536,B 2.4042,C 0.0611,E1 2.2707,E2 304.1247} C_DIS
LIN {X -111.9215,Y 73.4552,Z 187,A 147.6207,B 2.4043,C 0.0577,E1 2.2735,E2 305.9794} C_DIS
LIN {X -109.7274,Y 76.6945,Z 187,A 145.9766,B 2.4043,C 0.0539,E1 2.2761,E2 307.6186} C_DIS
LIN {X -107.8207,Y 79.3521,Z 187,A 144.4002,B 2.4045,C 0.0512,E1 2.2787,E2 309.2148} C_DIS
LIN {X -105.0388,Y 83.0004,Z 187,A 142.3071,B 2.4045,C 0.0473,E1 2.2823,E2 311.3216} C_DIS
LIN {X -102.7485,Y 85.8189,Z 187,A 140.6964,B 2.4045,C 0.0442,E1 2.2852,E2 312.9379} C_DIS
LIN {X -99.8704,Y 89.1516,Z 187,A 138.8083,B 2.4047,C 0.0403,E1 2.2887,E2 314.825} C_DIS
LIN {X -97.1593,Y 92.099,Z 187,A 137.0322,B 2.4047,C 0.0371,E1 2.2921,E2 316.6071} C_DIS
LIN {X -94.2563,Y 95.0675,Z 187,A 135.1673,B 2.4047,C 0.034,E1 2.2958,E2 318.481} C_DIS
LIN {X -91.5365,Y 97.6898,Z 187,A 133.3967,B 2.4047,C 0.0314,E1 2.2994,E2 320.2684} C_DIS
LIN {X -88.4885,Y 100.4585,Z 187,A 131.5472,B 2.4048,C 0.0285,E1 2.3033,E2 322.1267} C_DIS
LIN {X -84.9775,Y 103.4456,Z 187,A 129.4969,B 2.4048,C 0.0254,E1 2.3077,E2 324.1847} C_DIS
LIN {X -81.4708,Y 106.229,Z 187,A 127.5562,B 2.4048,C 0.0224,E1 2.3119,E2 326.1269} C_DIS
LIN {X -78.4145,Y 108.5046,Z 187,A 125.9723,B 2.4049,C 0.0197,E1 2.3155,E2 327.7042} C_DIS
LIN {X -75.7131,Y 110.4065,Z 187,A 124.513,B 2.4049,C 0.0177,E1 2.3189,E2 329.1677} C_DIS
LIN {X -72.9874,Y 112.2271,Z 187,A 122.9748,B 2.4049,C 0.0162,E1 2.3225,E2 330.7207} C_DIS
LIN {X -69.2418,Y 114.5759,Z 187,A 121.1169,B 2.4049,C 0.0135,E1 2.3269,E2 332.5734} C_DIS
LIN {X -66.418,Y 116.2356,Z 187,A 119.6775,B 2.4049,C 0.0118,E1 2.3304,E2 334.0162} C_DIS
LIN {X -63.5546,Y 117.8258,Z 187,A 118.1202,B 2.4049,C 0.0107,E1 2.3343,E2 335.5905} C_DIS
LIN {X -60.1851,Y 119.5811,Z 187,A 116.6024,B 2.4049,C 0.0084,E1 2.338,E2 337.0948} C_DIS
LIN {X -57.6836,Y 120.8061,Z 187,A 115.3485,B 2.4049,C 0.0073,E1 2.3412,E2 338.355} C_DIS
LIN {X -54.7049,Y 122.1839,Z 187,A 113.8885,B 2.4049,C 0.0061,E1 2.3449,E2 339.8205} C_DIS
LIN {X -51.6051,Y 123.5251,Z 187,A 112.4416,B 2.4049,C 0.0047,E1 2.3486,E2 341.2667} C_DIS
LIN {X -48.6009,Y 124.7377,Z 187,A 110.9407,B 2.4049,C 0.0039,E1 2.3526,E2 342.7799} C_DIS
LIN {X -45.0913,Y 126.0493,Z 187,A 109.3911,B 2.4049,C 0.0024,E1 2.3566,E2 344.3224} C_DIS
LIN {X -42.0027,Y 127.1118,Z 187,A 107.9713,B 2.4049,C 0.0015,E1 2.3604,E2 345.7439} C_DIS
LIN {X -38.855,Y 128.1092,Z 187,A 106.5371,B 2.4049,C 0.0006,E1 2.3642,E2 347.1797} C_DIS
LIN {X -35.702,Y 129.0235,Z 187,A 105.1144,B 2.4049,C -0.0002,E1 2.3681,E2 348.6036} C_DIS
LIN {X -32.5292,Y 129.8599,Z 187,A 103.695,B 2.4049,C -0.0009,E1 2.3719,E2 350.0241} C_DIS
LIN {X -29.3336,Y 130.6192,Z 187,A 102.2757,B 2.4049,C -0.0015,E1 2.3758,E2 351.4442} C_DIS
LIN {X -26.1055,Y 131.3029,Z 187,A 100.8549,B 2.4049,C -0.002,E1 2.3797,E2 352.8653} C_DIS
LIN {X -22.8798,Y 131.9039,Z 187,A 99.4444,B 2.4049,C -0.0025,E1 2.3836,E2 354.2758} C_DIS
LIN {X -19.6427,Y 132.4247,Z 187,A 98.0629,B 2.4049,C -0.0029,E1 2.3874,E2 355.6541} C_DIS
LIN {X -17.0133,Y 132.7867,Z 187,A 96.7575,B 2.4049,C -0.0024,E1 2.3911,E2 356.9783} C_DIS
LIN {X -13.1058,Y 133.229,Z 187,A 95.1865,B 2.4049,C -0.0031,E1 2.3954,E2 358.5357} C_DIS
LIN {X -9.8394,Y 133.5097,Z 187,A 93.7148,B 2.4049,C -0.0029,E1 2.3995,E2 360.0145} C_DIS
LIN {X -5.4232,Y 133.7621,Z 187,A 91.8916,B 2.4049,C -0.0032,E1 2.4046,E2 361.8289} C_DIS
LIN {X -1.6198,Y 133.8634,Z 187,A 90.3164,B 2.4049,C -0.0032,E1 2.409,E2 363.3974} C_DIS
LIN {X 1.6589,Y 133.8628,Z 187,A 88.8559,B 2.4049,C -0.0027,E1 2.4131,E2 364.8639} C_DIS
LIN {X 5.7591,Y 133.749,Z 187,A 86.9808,B 2.4049,C -0.0016,E1 2.4184,E2 366.752} C_DIS
LIN {X 10.3408,Y 133.4731,Z 187,A 85.0215,B 2.4049,C -0.0009,E1 2.4238,E2 368.71} C_DIS
LIN {X 14.2739,Y 133.1086,Z 187,A 83.5016,B 2.4049,C -0.0011,E1 2.428,E2 370.2096} C_DIS
LIN {X 17.5309,Y 132.7189,Z 187,A 82.0628,B 2.4049,C -0.0002,E1 2.432,E2 371.6519} C_DIS
LIN {X 20.7779,Y 132.2497,Z 187,A 80.7315,B 2.4049,C 0.0002,E1 2.4357,E2 372.9744} C_DIS
LIN {X 24.0101,Y 131.7016,Z 187,A 79.3486,B 2.4049,C 0.001,E1 2.4395,E2 374.3546} C_DIS
LIN {X 27.2489,Y 131.0703,Z 187,A 77.9575,B 2.4049,C 0.0019,E1 2.4433,E2 375.7428} C_DIS
LIN {X 30.4538,Y 130.3633,Z 187,A 76.5751,B 2.4049,C 0.0029,E1 2.447,E2 377.1223} C_DIS
LIN {X 33.6403,Y 129.5779,Z 187,A 75.1941,B 2.4049,C 0.0039,E1 2.4508,E2 378.5002} C_DIS
LIN {X 36.8063,Y 128.7147,Z 187,A 73.8146,B 2.4049,C 0.0051,E1 2.4545,E2 379.8765} C_DIS
LIN {X 39.95,Y 127.7741,Z 187,A 72.437,B 2.4049,C 0.0063,E1 2.4582,E2 381.2507} C_DIS
LIN {X 43.1044,Y 126.7446,Z 187,A 71.0483,B 2.4049,C 0.0076,E1 2.4618,E2 382.6354} C_DIS
LIN {X 46.1941,Y 125.6516,Z 187,A 69.5365,B 2.4049,C 0.0098,E1 2.4658,E2 384.1597} C_DIS
LIN {X 49.7139,Y 124.2988,Z 187,A 68.1029,B 2.4049,C 0.0105,E1 2.4695,E2 385.5719} C_DIS
LIN {X 52.7457,Y 123.043,Z 187,A 66.7353,B 2.4049,C 0.012,E1 2.473,E2 386.9351} C_DIS
LIN {X 55.7444,Y 121.7141,Z 187,A 65.3701,B 2.4049,C 0.0136,E1 2.4765,E2 388.2956} C_DIS
LIN {X 58.7119,Y 120.311,Z 187,A 64.0023,B 2.4049,C 0.0153,E1 2.4799,E2 389.6589} C_DIS
LIN {X 61.5765,Y 118.8714,Z 187,A 62.5542,B 2.4049,C 0.0177,E1 2.4836,E2 391.1158} C_DIS
LIN {X 65.555,Y 116.7245,Z 187,A 60.7122,B 2.4049,C 0.0199,E1 2.4881,E2 392.9468} C_DIS
LIN {X 68.8294,Y 114.8246,Z 187,A 59.2182,B 2.4049,C 0.0216,E1 2.4916,E2 394.426} C_DIS
LIN {X 71.6218,Y 113.1035,Z 187,A 57.7757,B 2.4049,C 0.0241,E1 2.4951,E2 395.8729} C_DIS
LIN {X 75.3174,Y 110.6772,Z 187,A 56.1262,B 2.4049,C 0.0256,E1 2.4988,E2 397.494} C_DIS
LIN {X 78.0206,Y 108.7882,Z 187,A 54.674,B 2.4049,C 0.0284,E1 2.5022,E2 398.9509} C_DIS
LIN {X 81.0712,Y 106.5346,Z 187,A 53.0599,B 2.4048,C 0.0312,E1 2.5058,E2 400.564} C_DIS
LIN {X 84.2962,Y 104.0015,Z 187,A 51.311,B 2.4048,C 0.0344,E1 2.5096,E2 402.3123} C_DIS
LIN {X 87.4422,Y 101.3702,Z 187,A 49.6381,B 2.4048,C 0.0372,E1 2.5131,E2 403.9756} C_DIS
LIN {X 90.5248,Y 98.6272,Z 187,A 47.9488,B 2.4047,C 0.0401,E1 2.5166,E2 405.6559} C_DIS
LIN {X 93.4972,Y 95.8146,Z 187,A 46.251,B 2.4047,C 0.0433,E1 2.52,E2 407.3477} C_DIS
LIN {X 96.3968,Y 92.8967,Z 187,A 44.6372,B 2.4046,C 0.0459,E1 2.5232,E2 408.9444} C_DIS
LIN {X 99.1964,Y 89.9007,Z 187,A 42.9005,B 2.4045,C 0.0495,E1 2.5264,E2 410.6792} C_DIS
LIN {X 102.0646,Y 86.6308,Z 187,A 41.1202,B 2.4045,C 0.053,E1 2.5297,E2 412.4501} C_DIS
LIN {X 104.871,Y 83.2116,Z 187,A 39.3197,B 2.4043,C 0.0565,E1 2.5328,E2 414.2401} C_DIS
LIN {X 107.5276,Y 79.7493,Z 187,A 37.6262,B 2.4043,C 0.0595,E1 2.5356,E2 415.9132} C_DIS
LIN {X 109.4613,Y 77.0733,Z 187,A 36.2826,B 2.4042,C 0.0623,E1 2.5378,E2 417.2489} C_DIS
LIN {X 111.3158,Y 74.3697,Z 187,A 34.9492,B 2.4042,C 0.0651,E1 2.5399,E2 418.5743} C_DIS
LIN {X 113.3692,Y 71.201,Z 187,A 33.2867,B 2.404,C 0.0694,E1 2.5424,E2 420.2428} C_DIS
LIN {X 115.4061,Y 67.8489,Z 187,A 31.8756,B 2.404,C 0.0714,E1 2.5444,E2 421.6223} C_DIS
LIN {X 117.0415,Y 64.9875,Z 187,A 30.4764,B 2.4038,C 0.0748,E1 2.5463,E2 423.0206} C_DIS
LIN {X 118.829,Y 61.6571,Z 187,A 28.9311,B 2.4038,C 0.0783,E1 2.5483,E2 424.5577} C_DIS
LIN {X 120.0948,Y 59.1503,Z 187,A 27.7974,B 2.4036,C 0.0808,E1 2.5497,E2 425.6835} C_DIS
LIN {X 121.507,Y 56.1922,Z 187,A 26.4676,B 2.4036,C 0.0839,E1 2.5513,E2 427.005} C_DIS
LIN {X 122.8467,Y 53.1998,Z 187,A 25.1379,B 2.4034,C 0.0869,E1 2.5528,E2 428.3264} C_DIS
LIN {X 124.1128,Y 50.1755,Z 187,A 23.796,B 2.4034,C 0.0901,E1 2.5542,E2 429.6614} C_DIS
LIN {X 125.4862,Y 46.6355,Z 187,A 22.2694,B 2.4032,C 0.0936,E1 2.5557,E2 431.1768} C_DIS
LIN {X 126.5892,Y 43.5525,Z 187,A 20.9412,B 2.403,C 0.0968,E1 2.5569,E2 432.4967} C_DIS
LIN {X 127.6193,Y 40.4348,Z 187,A 19.6113,B 2.403,C 0.0999,E1 2.5581,E2 433.818} C_DIS
LIN {X 128.5758,Y 37.282,Z 187,A 18.2794,B 2.4028,C 0.1031,E1 2.5591,E2 435.1411} C_DIS
LIN {X 129.4514,Y 34.1182,Z 187,A 16.9519,B 2.4026,C 0.1063,E1 2.5601,E2 436.4598} C_DIS
LIN {X 130.2489,Y 30.9354,Z 187,A 15.6255,B 2.4026,C 0.1095,E1 2.5609,E2 437.7773} C_DIS
LIN {X 130.9689,Y 27.7314,Z 187,A 14.2988,B 2.4024,C 0.1128,E1 2.5617,E2 439.0951} C_DIS
LIN {X 131.613,Y 24.4956,Z 187,A 12.9686,B 2.4022,C 0.116,E1 2.5624,E2 440.416} C_DIS
LIN {X 132.1744,Y 21.2636,Z 187,A 11.6232,B 2.402,C 0.1194,E1 2.563,E2 441.7551} C_DIS
LIN {X 132.5863,Y 18.5116,Z 187,A 10.4286,B 2.4019,C 0.1228,E1 2.5635,E2 442.9507} C_DIS
LIN {X 133.0572,Y 14.7509,Z 187,A 8.9684,B 2.4017,C 0.1259,E1 2.564,E2 444.3919} C_DIS
LIN {X 133.3504,Y 11.8157,Z 187,A 7.6969,B 2.4015,C 0.1296,E1 2.5643,E2 445.6653} C_DIS
LIN {X 133.651,Y 7.7028,Z 187,A 5.9856,B 2.4013,C 0.1341,E1 2.5646,E2 447.371} C_DIS
LIN {X 133.8183,Y 3.7867,Z 187,A 4.4734,B 2.4011,C 0.1374,E1 2.5648,E2 448.8637} C_DIS
LIN {X 133.8732,Y 0.0844,Z 187,A 3.0145,B 2.4009,C 0.1408,E1 2.5648,E2 450.3081} C_DIS
LIN {X 133.8437,Y -2.8074,Z 187,A 1.76,B 2.4007,C 0.1444,E1 2.5648,E2 451.5654} C_DIS
LIN {X 133.7104,Y -6.5735,Z 187,A 0.3693,B 2.4005,C 0.1471,E1 2.5646,E2 452.9296} C_DIS
LIN {X 133.4731,Y -10.3409,Z 187,A -1.2736,B 2.4002,C 0.1519,E1 2.5643,E2 454.5769} C_DIS
LIN {X 133.1085,Y -14.2748,Z 187,A -2.7753,B 2.4,C 0.155,E1 2.5639,E2 456.0561} C_DIS
LIN {X 132.7188,Y -17.5314,Z 187,A -4.1481,B 2.3998,C 0.1587,E1 2.5634,E2 457.426} C_DIS
LIN {X 132.2497,Y -20.7781,Z 187,A -5.4218,B 2.3996,C 0.1615,E1 2.5629,E2 458.6844} C_DIS
LIN {X 131.7016,Y -24.0101,Z 187,A -6.7462,B 2.3993,C 0.1648,E1 2.5622,E2 459.9999} C_DIS
LIN {X 131.0739,Y -27.2312,Z 187,A -8.0735,B 2.3991,C 0.168,E1 2.5615,E2 461.3186} C_DIS
LIN {X 130.368,Y -30.433,Z 187,A -9.4009,B 2.3989,C 0.1713,E1 2.5607,E2 462.6375} C_DIS
LIN {X 129.5782,Y -33.6393,Z 187,A -10.7376,B 2.3987,C 0.1745,E1 2.5598,E2 463.9655} C_DIS
LIN {X 128.7143,Y -36.8075,Z 187,A -12.0682,B 2.3984,C 0.1777,E1 2.5588,E2 465.2877} C_DIS
LIN {X 127.7737,Y -39.9512,Z 187,A -13.4304,B 2.3982,C 0.1812,E1 2.5577,E2 466.6456} C_DIS
LIN {X 126.7325,Y -43.139,Z 187,A -14.7489,B 2.3979,C 0.1841,E1 2.5565,E2 467.9504} C_DIS
LIN {X 125.6502,Y -46.1978,Z 187,A -16.1085,B 2.3977,C 0.1875,E1 2.5552,E2 469.3074} C_DIS
LIN {X 124.3062,Y -49.6957,Z 187,A -17.5956,B 2.3974,C 0.1908,E1 2.5537,E2 470.7809} C_DIS
LIN {X 123.0411,Y -52.7501,Z 187,A -18.9294,B 2.3972,C 0.1938,E1 2.5523,E2 472.1055} C_DIS
LIN {X 121.7109,Y -55.7513,Z 187,A -20.26,B 2.3969,C 0.1969,E1 2.5508,E2 473.4277} C_DIS
LIN {X 120.3076,Y -58.7189,Z 187,A -21.5049,B 2.3967,C 0.1992,E1 2.5493,E2 474.6533} C_DIS
LIN {X 119.0419,Y -61.2442,Z 187,A -22.7502,B 2.3965,C 0.2026,E1 2.5477,E2 475.9042} C_DIS
LIN {X 117.2726,Y -64.5702,Z 187,A -24.2695,B 2.3962,C 0.2059,E1 2.5457,E2 477.4129} C_DIS
LIN {X 115.8317,Y -67.12,Z 187,A -25.5175,B 2.3959,C 0.209,E1 2.544,E2 478.6612} C_DIS
LIN {X 113.9741,Y -70.2284,Z 187,A -26.9423,B 2.3957,C 0.2118,E1 2.5419,E2 480.0713} C_DIS
LIN {X 111.9523,Y -73.4085,Z 187,A -28.5854,B 2.3953,C 0.2159,E1 2.5394,E2 481.7195} C_DIS
LIN {X 109.7578,Y -76.6506,Z 187,A -30.0708,B 2.3951,C 0.2184,E1 2.5371,E2 483.1819} C_DIS
LIN {X 107.8278,Y -79.3424,Z 187,A -31.4059,B 2.3948,C 0.221,E1 2.535,E2 484.5075} C_DIS
LIN {X 105.5303,Y -82.3746,Z 187,A -33.0881,B 2.3944,C 0.2252,E1 2.5321,E2 486.198} C_DIS
LIN {X 102.9602,Y -85.5646,Z 187,A -34.6814,B 2.3942,C 0.2279,E1 2.5293,E2 487.7721} C_DIS
LIN {X 100.2929,Y -88.6757,Z 187,A -36.4163,B 2.3938,C 0.2316,E1 2.5261,E2 489.5058} C_DIS
LIN {X 97.5219,Y -91.7147,Z 187,A -38.1098,B 2.3935,C 0.2349,E1 2.5229,E2 491.1921} C_DIS
LIN {X 94.5802,Y -94.7456,Z 187,A -39.8658,B 2.3932,C 0.2383,E1 2.5195,E2 492.943} C_DIS
LIN {X 91.5364,Y -97.6899,Z 187,A -41.5907,B 2.3929,C 0.2413,E1 2.516,E2 494.658} C_DIS
LIN {X 88.2501,Y -100.6681,Z 187,A -43.397,B 2.3926,C 0.2444,E1 2.5123,E2 496.4539} C_DIS
LIN {X 84.9196,Y -103.4929,Z 187,A -45.1975,B 2.3922,C 0.2474,E1 2.5084,E2 498.247} C_DIS
LIN {X 81.5182,Y -106.1927,Z 187,A -46.9841,B 2.3919,C 0.2504,E1 2.5045,E2 500.0257} C_DIS
LIN {X 78.0167,Y -108.791,Z 187,A -48.8013,B 2.3916,C 0.2533,E1 2.5004,E2 501.838} C_DIS
LIN {X 74.3695,Y -111.3159,Z 187,A -50.5442,B 2.3914,C 0.2554,E1 2.4964,E2 503.5622} C_DIS
LIN {X 71.072,Y -113.4504,Z 187,A -52.254,B 2.3911,C 0.2584,E1 2.4924,E2 505.2769} C_DIS
LIN {X 67.7935,Y -115.4387,Z 187,A -53.7192,B 2.3909,C 0.2598,E1 2.4889,E2 506.7205} C_DIS
LIN {X 64.9794,Y -117.046,Z 187,A -55.0606,B 2.3907,C 0.2616,E1 2.4856,E2 508.0569} C_DIS
LIN {X 61.6392,Y -118.8384,Z 187,A -56.6479,B 2.3905,C 0.2637,E1 2.4817,E2 509.6408} C_DIS
LIN {X 59.1543,Y -120.0928,Z 187,A -57.7979,B 2.3904,C 0.2651,E1 2.4789,E2 510.7862} C_DIS
LIN {X 56.1944,Y -121.506,Z 187,A -59.1617,B 2.3902,C 0.2667,E1 2.4754,E2 512.1458} C_DIS
LIN {X 53.2041,Y -122.8448,Z 187,A -60.5268,B 2.39,C 0.2683,E1 2.4719,E2 513.5071} C_DIS
LIN {X 50.1747,Y -124.1131,Z 187,A -61.8962,B 2.3898,C 0.2698,E1 2.4684,E2 514.8727} C_DIS
LIN {X 46.6511,Y -125.4804,Z 187,A -63.4759,B 2.3896,C 0.2714,E1 2.4643,E2 516.4486} C_DIS
LIN {X 43.5621,Y -126.5859,Z 187,A -64.8489,B 2.3895,C 0.2728,E1 2.4607,E2 517.8184} C_DIS
LIN {X 40.4305,Y -127.6207,Z 187,A -66.2292,B 2.3893,C 0.274,E1 2.457,E2 519.1955} C_DIS
LIN {X 37.2771,Y -128.5772,Z 187,A -67.608,B 2.3893,C 0.2752,E1 2.4533,E2 520.5712} C_DIS
LIN {X 34.114,Y -129.4526,Z 187,A -68.9849,B 2.3891,C 0.2763,E1 2.4496,E2 521.9453} C_DIS
LIN {X 30.9302,Y -130.2502,Z 187,A -70.3634,B 2.389,C 0.2774,E1 2.4459,E2 523.3212} C_DIS
LIN {X 27.73,Y -130.9692,Z 187,A -71.7431,B 2.3888,C 0.2783,E1 2.4421,E2 524.6987} C_DIS
LIN {X 24.484,Y -131.6153,Z 187,A -73.1334,B 2.3888,C 0.2792,E1 2.4383,E2 526.0863} C_DIS
LIN {X 21.2534,Y -132.1761,Z 187,A -74.512,B 2.3887,C 0.28,E1 2.4345,E2 527.4626} C_DIS
LIN {X 18.5021,Y -132.5876,Z 187,A -75.787,B 2.3885,C 0.2812,E1 2.4309,E2 528.7493} C_DIS
LIN {X 14.7566,Y -133.0566,Z 187,A -77.3187,B 2.3885,C 0.2815,E1 2.4267,E2 530.2708} C_DIS
LIN {X 11.4614,Y -133.3803,Z 187,A -78.7069,B 2.3885,C 0.282,E1 2.4228,E2 531.6561} C_DIS
LIN {X 7.6886,Y -133.6519,Z 187,A -80.4502,B 2.3883,C 0.2834,E1 2.4179,E2 533.4164} C_DIS
LIN {X 3.7763,Y -133.8186,Z 187,A -82.0377,B 2.3883,C 0.2834,E1 2.4135,E2 534.9933} C_DIS
LIN {X 0.9691,Y -133.8678,Z 187,A -82.8688,B 2.3885,C 0.2815,E1 2.4113,E2 535.7764} C_DIS
Enddeposition()
LIN {X 0.9691,Y -133.8678,Z 187,A -82.8688,B 2.3885,C 0.2815,E1 2.4113,E2 535.7764} C_DIS
Startdeposition()
$VEL.CP = VEL_PRINT
LIN {X 1.3335,Y -134.7662,Z 187,A -82.2771,B 2.3887,C 0.2802,E1 2.4131,E2 535.1563} C_DIS
LIN {X 5.3795,Y -134.6642,Z 187,A -80.628,B 2.3887,C 0.2802,E1 2.4177,E2 533.5158} C_DIS
LIN {X 8.7448,Y -134.4882,Z 187,A -78.8627,B 2.389,C 0.2776,E1 2.4228,E2 531.7054} C_DIS
LIN {X 12.4296,Y -134.1978,Z 187,A -77.5253,B 2.389,C 0.2783,E1 2.4264,E2 530.3985} C_DIS
LIN {X 17.0558,Y -133.6886,Z 187,A -75.582,B 2.389,C 0.2775,E1 2.4318,E2 528.4588} C_DIS
LIN {X 21.7836,Y -132.9998,Z 187,A -73.6929,B 2.389,C 0.2771,E1 2.437,E2 526.5875} C_DIS
LIN {X 26.8208,Y -132.0755,Z 187,A -71.5846,B 2.3892,C 0.276,E1 2.4428,E2 524.487} C_DIS
LIN {X 30.1541,Y -131.3546,Z 187,A -70.1545,B 2.3893,C 0.2749,E1 2.4466,E2 523.0587} C_DIS
LIN {X 33.5056,Y -130.5403,Z 187,A -68.6105,B 2.3895,C 0.2731,E1 2.4509,E2 521.5035} C_DIS
LIN {X 37.6683,Y -129.4002,Z 187,A -66.9104,B 2.3896,C 0.2723,E1 2.4554,E2 519.8201} C_DIS
LIN {X 40.7728,Y -128.4558,Z 187,A -65.6069,B 2.3897,C 0.2714,E1 2.4589,E2 518.5258} C_DIS
LIN {X 43.3623,Y -127.6074,Z 187,A -64.2764,B 2.39,C 0.269,E1 2.4625,E2 517.1718} C_DIS
LIN {X 47.0033,Y -126.3092,Z 187,A -62.8201,B 2.39,C 0.2684,E1 2.4662,E2 515.7392} C_DIS
LIN {X 49.7898,Y -125.2382,Z 187,A -61.4986,B 2.3903,C 0.2665,E1 2.4697,E2 514.4099} C_DIS
LIN {X 53.4423,Y -123.722,Z 187,A -60.0358,B 2.3903,C 0.2659,E1 2.4734,E2 512.9749} C_DIS
LIN {X 55.8466,Y -122.658,Z 187,A -58.7162,B 2.3907,C 0.263,E1 2.4768,E2 511.6278} C_DIS
LIN {X 59.0063,Y -121.169,Z 187,A -57.2998,B 2.3908,C 0.2614,E1 2.4804,E2 510.2195} C_DIS
LIN {X 64.2612,Y -118.4667,Z 187,A -55.0948,B 2.391,C 0.26,E1 2.4857,E2 508.0534} C_DIS
LIN {X 69.6737,Y -115.3661,Z 187,A -51.9418,B 2.3918,C 0.2522,E1 2.4935,E2 504.8321} C_DIS
LIN {X 73.2965,Y -113.099,Z 187,A -50.5387,B 2.3918,C 0.2522,E1 2.4967,E2 503.4825} C_DIS
LIN {X 77.1527,Y -110.5045,Z 187,A -48.7059,B 2.3921,C 0.2499,E1 2.5009,E2 501.6672} C_DIS
LIN {X 80.8649,Y -107.8182,Z 187,A -46.7589,B 2.3924,C 0.2464,E1 2.5052,E2 499.7189} C_DIS
LIN {X 84.1219,Y -105.2963,Z 187,A -45.1317,B 2.3927,C 0.2441,E1 2.5088,E2 498.1068} C_DIS
LIN {X 87.6335,Y -102.3928,Z 187,A -43.1864,B 2.393,C 0.2403,E1 2.513,E2 496.1589} C_DIS
LIN {X 90.1847,Y -100.1529,Z 187,A -41.8109,B 2.3933,C 0.238,E1 2.5158,E2 494.7912} C_DIS
LIN {X 93.5123,Y -97.0531,Z 187,A -39.996,B 2.3936,C 0.2349,E1 2.5195,E2 492.9904} C_DIS
LIN {X 95.6414,Y -94.9552,Z 187,A -38.6572,B 2.3939,C 0.2318,E1 2.5221,E2 491.6416} C_DIS
LIN {X 99.1475,Y -91.2882,Z 187,A -36.9271,B 2.394,C 0.2305,E1 2.5253,E2 489.9659} C_DIS
LIN {X 101.1526,Y -89.0617,Z 187,A -35.4877,B 2.3944,C 0.2264,E1 2.528,E2 488.5038} C_DIS
LIN {X 104.0038,Y -85.715,Z 187,A -33.7177,B 2.3947,C 0.223,E1 2.5312,E2 486.7454} C_DIS
LIN {X 106.7754,Y -82.2371,Z 187,A -31.8735,B 2.3951,C 0.2191,E1 2.5344,E2 484.9057} C_DIS
LIN {X 109.5011,Y -78.5704,Z 187,A -29.7504,B 2.3956,C 0.213,E1 2.5379,E2 482.7575} C_DIS
LIN {X 111.7217,Y -75.3794,Z 187,A -28.5452,B 2.3956,C 0.2127,E1 2.5397,E2 481.6095} C_DIS
LIN {X 113.833,Y -72.1516,Z 187,A -26.9942,B 2.3959,C 0.2095,E1 2.542,E2 480.0688} C_DIS
LIN {X 115.9464,Y -68.7045,Z 187,A -25.3603,B 2.3962,C 0.2059,E1 2.5444,E2 478.4446} C_DIS
LIN {X 118.1529,Y -64.8365,Z 187,A -23.1447,B 2.3969,C 0.1985,E1 2.5474,E2 476.1855} C_DIS
LIN {X 120.0029,Y -61.3397,Z 187,A -22.0424,B 2.3969,C 0.1991,E1 2.5488,E2 475.1572} C_DIS
LIN {X 121.5819,Y -58.1468,Z 187,A -20.5327,B 2.3971,C 0.1952,E1 2.5506,E2 473.647} C_DIS
LIN {X 122.913,Y -55.2782,Z 187,A -19.343,B 2.3973,C 0.193,E1 2.552,E2 472.4762} C_DIS
LIN {X 124.0466,Y -52.6908,Z 187,A -18.1386,B 2.3976,C 0.1898,E1 2.5533,E2 471.2705} C_DIS
LIN {X 125.8527,Y -48.2158,Z 187,A -15.1072,B 2.3986,C 0.1762,E1 2.5565,E2 468.1102} C_DIS
LIN {X 128.4064,Y -40.9275,Z 187,A -13.184,B 2.3984,C 0.1788,E1 2.558,E2 466.3611} C_DIS
LIN {X 129.2725,Y -38.1043,Z 187,A -12.0616,B 2.3986,C 0.1765,E1 2.5589,E2 465.2549} C_DIS
LIN {X 130.1625,Y -34.9435,Z 187,A -10.5492,B 2.3989,C 0.1717,E1 2.56,E2 463.7265} C_DIS
LIN {X 130.9415,Y -31.9015,Z 187,A -9.2545,B 2.3992,C 0.1684,E1 2.5609,E2 462.436} C_DIS
LIN {X 131.7738,Y -28.2664,Z 187,A -7.807,B 2.3994,C 0.1652,E1 2.5617,E2 461.005} C_DIS
LIN {X 132.5575,Y -24.3345,Z 187,A -6.1682,B 2.3997,C 0.161,E1 2.5626,E2 459.3735} C_DIS
LIN {X 133.0827,Y -21.278,Z 187,A -4.8134,B 2.3999,C 0.1571,E1 2.5632,E2 458.0132} C_DIS
LIN {X 133.6547,Y -17.3139,Z 187,A -3.2943,B 2.4001,C 0.1539,E1 2.5638,E2 456.5163} C_DIS
LIN {X 134.282,Y -11.4764,Z 187,A -0.9218,B 2.4005,C 0.1479,E1 2.5644,E2 454.1578} C_DIS
LIN {X 134.5713,Y -7.368,Z 187,A 0.7395,B 2.4008,C 0.1438,E1 2.5647,E2 452.5069} C_DIS
LIN {X 134.7414,Y -2.932,Z 187,A 2.3947,B 2.401,C 0.1404,E1 2.5649,E2 450.8799} C_DIS
LIN {X 134.7715,Y 0.3542,Z 187,A 3.8919,B 2.4012,C 0.1356,E1 2.5649,E2 449.3692} C_DIS
LIN {X 134.6798,Y 4.9794,Z 187,A 5.6557,B 2.4015,C 0.1318,E1 2.5647,E2 447.6298} C_DIS
LIN {X 134.46,Y 9.1784,Z 187,A 7.5155,B 2.4018,C 0.1262,E1 2.5644,E2 445.7598} C_DIS
LIN {X 134.027,Y 14.1482,Z 187,A 9.1133,B 2.4018,C 0.1246,E1 2.564,E2 444.2265} C_DIS
LIN {X 133.6768,Y 17.1457,Z 187,A 10.5372,B 2.4021,C 0.1199,E1 2.5635,E2 442.7843} C_DIS
LIN {X 133.1845,Y 20.6202,Z 187,A 11.9368,B 2.4023,C 0.1165,E1 2.563,E2 441.3955} C_DIS
LIN {X 132.5397,Y 24.4337,Z 187,A 13.6033,B 2.4025,C 0.1117,E1 2.5621,E2 439.7254} C_DIS
LIN {X 131.7915,Y 28.1841,Z 187,A 15.0375,B 2.4026,C 0.1089,E1 2.5613,E2 438.3141} C_DIS
LIN {X 131.0112,Y 31.6122,Z 187,A 16.3304,B 2.4027,C 0.1064,E1 2.5605,E2 437.0457} C_DIS
LIN {X 130.3719,Y 34.158,Z 187,A 17.4147,B 2.4028,C 0.1036,E1 2.5598,E2 435.9648} C_DIS
LIN {X 129.5562,Y 37.1355,Z 187,A 18.8716,B 2.403,C 0.0989,E1 2.5587,E2 434.4893} C_DIS
LIN {X 128.4813,Y 40.693,Z 187,A 20.2898,B 2.4032,C 0.0959,E1 2.5575,E2 433.0904} C_DIS
LIN {X 127.0451,Y 44.9821,Z 187,A 22.0268,B 2.4033,C 0.0923,E1 2.556,E2 431.3757} C_DIS
LIN {X 126.1589,Y 47.4044,Z 187,A 23.4713,B 2.4035,C 0.0866,E1 2.5545,E2 429.8876} C_DIS
LIN {X 124.7093,Y 51.1021,Z 187,A 24.8659,B 2.4035,C 0.0845,E1 2.5531,E2 428.5289} C_DIS
LIN {X 123.0123,Y 55.0562,Z 187,A 26.4351,B 2.4037,C 0.0819,E1 2.5513,E2 426.991} C_DIS
LIN {X 121.7902,Y 57.7109,Z 187,A 27.7452,B 2.4038,C 0.0782,E1 2.5498,E2 425.6721} C_DIS
LIN {X 119.7342,Y 61.8675,Z 187,A 29.6084,B 2.4039,C 0.074,E1 2.5474,E2 423.8217} C_DIS
LIN {X 117.5745,Y 65.8789,Z 187,A 31.1626,B 2.4039,C 0.0722,E1 2.5454,E2 422.3137} C_DIS
LIN {X 116.1932,Y 68.2853,Z 187,A 32.53,B 2.4041,C 0.0678,E1 2.5435,E2 420.923} C_DIS
LIN {X 113.9281,Y 72.001,Z 187,A 34.1807,B 2.4041,C 0.0649,E1 2.5411,E2 419.2962} C_DIS
LIN {X 111.9225,Y 75.0814,Z 187,A 35.7421,B 2.4043,C 0.0612,E1 2.5387,E2 417.7346} C_DIS
LIN {X 109.4673,Y 78.6177,Z 187,A 37.5239,B 2.4043,C 0.0572,E1 2.5358,E2 415.9582} C_DIS
LIN {X 106.8369,Y 82.1569,Z 187,A 39.3236,B 2.4045,C 0.0535,E1 2.5328,E2 414.1672} C_DIS
LIN {X 104.0619,Y 85.6448,Z 187,A 41.1432,B 2.4045,C 0.0498,E1 2.5296,E2 412.3563} C_DIS
LIN {X 101.1304,Y 89.0867,Z 187,A 42.9771,B 2.4046,C 0.0463,E1 2.5262,E2 410.5328} C_DIS
LIN {X 97.9822,Y 92.5378,Z 187,A 44.6141,B 2.4046,C 0.0446,E1 2.5232,E2 408.9377} C_DIS
LIN {X 95.4781,Y 95.1195,Z 187,A 46.2681,B 2.4047,C 0.0405,E1 2.52,E2 407.2685} C_DIS
LIN {X 92.4558,Y 98.0596,Z 187,A 48.342,B 2.4048,C 0.0348,E1 2.5157,E2 405.1603} C_DIS
LIN {X 89.5581,Y 100.7137,Z 187,A 49.628,B 2.4048,C 0.0344,E1 2.5131,E2 403.9207} C_DIS
LIN {X 86.4295,Y 103.4106,Z 187,A 51.2995,B 2.4048,C 0.0316,E1 2.5096,E2 402.2592} C_DIS
LIN {X 83.0394,Y 106.1521,Z 187,A 53.1536,B 2.4049,C 0.0282,E1 2.5055,E2 400.405} C_DIS
LIN {X 79.5585,Y 108.7855,Z 187,A 54.8885,B 2.4049,C 0.0257,E1 2.5016,E2 398.6846} C_DIS
LIN {X 76.1449,Y 111.2013,Z 187,A 56.6158,B 2.4049,C 0.023,E1 2.4977,E2 396.9633} C_DIS
LIN {X 72.8618,Y 113.3798,Z 187,A 58.24,B 2.4049,C 0.0206,E1 2.4939,E2 395.3453} C_DIS
LIN {X 69.0514,Y 115.7396,Z 187,A 60.0679,B 2.405,C 0.0181,E1 2.4895,E2 393.5267} C_DIS
LIN {X 66.0975,Y 117.4516,Z 187,A 61.8552,B 2.405,C 0.0137,E1 2.4851,E2 391.6994} C_DIS
LIN {X 62.4995,Y 119.4029,Z 187,A 63.08,B 2.405,C 0.0146,E1 2.4822,E2 390.5362} C_DIS
LIN {X 59.618,Y 120.8673,Z 187,A 64.4034,B 2.405,C 0.013,E1 2.4789,E2 389.219} C_DIS
LIN {X 56.9479,Y 122.1488,Z 187,A 65.5999,B 2.405,C 0.0118,E1 2.4759,E2 388.0302} C_DIS
LIN {X 53.6701,Y 123.6235,Z 187,A 67.1363,B 2.405,C 0.0098,E1 2.472,E2 386.493} C_DIS
LIN {X 50.8457,Y 124.8126,Z 187,A 68.2669,B 2.405,C 0.0093,E1 2.4691,E2 385.383} C_DIS
LIN {X 48.0466,Y 125.9184,Z 187,A 69.7828,B 2.405,C 0.0063,E1 2.4651,E2 383.8395} C_DIS
LIN {X 44.2408,Y 127.3028,Z 187,A 71.3698,B 2.405,C 0.0053,E1 2.4609,E2 382.2686} C_DIS
LIN {X 41.0729,Y 128.3599,Z 187,A 72.6648,B 2.405,C 0.0046,E1 2.4575,E2 380.9887} C_DIS
LIN {X 38.2925,Y 129.2174,Z 187,A 73.8622,B 2.405,C 0.0036,E1 2.4543,E2 379.7962} C_DIS
LIN {X 35.2553,Y 130.0793,Z 187,A 75.3085,B 2.405,C 0.0018,E1 2.4504,E2 378.338} C_DIS
LIN {X 31.716,Y 130.9862,Z 187,A 76.831,B 2.405,C 0.0007,E1 2.4463,E2 376.8195} C_DIS
LIN {X 27.4388,Y 131.9497,Z 187,A 78.7055,B 2.405,C -0.0008,E1 2.4412,E2 374.9444} C_DIS
LIN {X 23.703,Y 132.6705,Z 187,A 80.2149,B 2.405,C -0.0012,E1 2.437,E2 373.4481} C_DIS
LIN {X 19.7877,Y 133.3128,Z 187,A 82.0021,B 2.405,C -0.0028,E1 2.4321,E2 371.6498} C_DIS
LIN {X 15.9102,Y 133.829,Z 187,A 83.565,B 2.405,C -0.0031,E1 2.4278,E2 370.0991} C_DIS
LIN {X 10.8412,Y 134.3356,Z 187,A 85.6303,B 2.405,C -0.0035,E1 2.422,E2 368.0465} C_DIS
LIN {X 7.2553,Y 134.5769,Z 187,A 87.0433,B 2.405,C -0.0034,E1 2.4181,E2 366.6476} C_DIS
LIN {X 4.5477,Y 134.6966,Z 187,A 88.4003,B 2.405,C -0.0048,E1 2.4143,E2 365.2669} C_DIS
LIN {X 0.8047,Y 134.7692,Z 187,A 90.0446,B 2.405,C -0.0054,E1 2.4097,E2 363.617} C_DIS
LIN {X -4.0504,Y 134.711,Z 187,A 92.003,B 2.405,C -0.0051,E1 2.4042,E2 361.672} C_DIS
LIN {X -8.1337,Y 134.5259,Z 187,A 93.7908,B 2.405,C -0.0054,E1 2.3992,E2 359.8791} C_DIS
LIN {X -12.6579,Y 134.1758,Z 187,A 96.0445,B 2.405,C -0.0068,E1 2.3928,E2 357.5879} C_DIS
LIN {X -16.5526,Y 133.7523,Z 187,A 97.3725,B 2.405,C -0.0049,E1 2.3892,E2 356.3007} C_DIS
LIN {X -20.3891,Y 133.2203,Z 187,A 98.9759,B 2.405,C -0.0043,E1 2.3848,E2 354.7031} C_DIS
LIN {X -23.8355,Y 132.6468,Z 187,A 100.4655,B 2.405,C -0.0038,E1 2.3807,E2 353.2137} C_DIS
LIN {X -27.7854,Y 131.8776,Z 187,A 102.2954,B 2.405,C -0.0038,E1 2.3757,E2 351.3708} C_DIS
LIN {X -31.2253,Y 131.1045,Z 187,A 103.7062,B 2.405,C -0.0026,E1 2.3718,E2 349.9712} C_DIS
LIN {X -34.0194,Y 130.4089,Z 187,A 104.9461,B 2.405,C -0.002,E1 2.3685,E2 348.7301} C_DIS
LIN {X -37.659,Y 129.4029,Z 187,A 106.5512,B 2.405,C -0.001,E1 2.3642,E2 347.1258} C_DIS
LIN {X -43.9472,Y 127.4046,Z 187,A 109.1632,B 2.405,C 0.0018,E1 2.3573,E2 344.5383} C_DIS
LIN {X -50.6169,Y 124.9048,Z 187,A 112.9023,B 2.405,C 0.0015,E1 2.3473,E2 340.7173} C_DIS
LIN {X -54.2583,Y 123.3692,Z 187,A 114.3565,B 2.405,C 0.0041,E1 2.3436,E2 339.2911} C_DIS
LIN {X -57.6494,Y 121.8195,Z 187,A 115.7278,B 2.405,C 0.0065,E1 2.3402,E2 337.9459} C_DIS
LIN {X -60.6856,Y 120.3359,Z 187,A 117.5612,B 2.405,C 0.0066,E1 2.3355,E2 336.0666} C_DIS
LIN {X -65.4838,Y 117.7951,Z 187,A 119.7188,B 2.405,C 0.01,E1 2.3303,E2 333.9284} C_DIS
LIN {X -68.7893,Y 115.8959,Z 187,A 121.388,B 2.405,C 0.0119,E1 2.3262,E2 332.2545} C_DIS
LIN {X -72.245,Y 113.7741,Z 187,A 123.1145,B 2.405,C 0.0142,E1 2.3221,E2 330.5289} C_DIS
LIN {X -74.6135,Y 112.2348,Z 187,A 124.5977,B 2.405,C 0.015,E1 2.3186,E2 329.0129} C_DIS
LIN {X -78.3532,Y 109.6564,Z 187,A 126.2294,B 2.405,C 0.0189,E1 2.3149,E2 327.418} C_DIS
LIN {X -84.4158,Y 105.0609,Z 187,A 130.2275,B 2.405,C 0.0217,E1 2.3059,E2 323.3314} C_DIS
LIN {X -87.7769,Y 102.2694,Z 187,A 131.7362,B 2.405,C 0.026,E1 2.3028,E2 321.8657} C_DIS
LIN {X -91.1408,Y 99.283,Z 187,A 133.6822,B 2.4049,C 0.0293,E1 2.2987,E2 319.9171} C_DIS
LIN {X -94.0944,Y 96.4891,Z 187,A 135.4417,B 2.4049,C 0.0324,E1 2.2952,E2 318.1551} C_DIS
LIN {X -97.7134,Y 92.8221,Z 187,A 137.8147,B 2.4049,C 0.0361,E1 2.2905,E2 315.7619} C_DIS
LIN {X -102.514,Y 87.4902,Z 187,A 140.959,B 2.4047,C 0.0421,E1 2.2847,E2 312.6086} C_DIS
LIN {X -106.2845,Y 82.8704,Z 187,A 143.6656,B 2.4047,C 0.047,E1 2.2799,E2 309.8834} C_DIS
LIN {X -108.8124,Y 79.5218,Z 187,A 145.4497,B 2.4045,C 0.0509,E1 2.2769,E2 308.1005} C_DIS
LIN {X -111.201,Y 76.1453,Z 187,A 147.9643,B 2.4045,C 0.053,E1 2.2728,E2 305.4956} C_DIS
LIN {X -114.0516,Y 71.8053,Z 187,A 149.5837,B 2.4043,C 0.0596,E1 2.2705,E2 303.9492} C_DIS
LIN {X -116.0163,Y 68.5865,Z 187,A 151.2982,B 2.4043,C 0.0631,E1 2.268,E2 302.2224} C_DIS
LIN {X -118.0441,Y 65.034,Z 187,A 153.1317,B 2.4041,C 0.0671,E1 2.2655,E2 300.3787} C_DIS
LIN {X -119.9195,Y 61.5034,Z 187,A 154.9056,B 2.4041,C 0.0711,E1 2.2632,E2 298.597} C_DIS
LIN {X -121.244,Y 58.854,Z 187,A 156.4209,B 2.4039,C 0.0736,E1 2.2613,E2 297.0517} C_DIS
LIN {X -123.3822,Y 54.2282,Z 187,A 158.6493,B 2.4038,C 0.079,E1 2.2587,E2 294.8173} C_DIS
LIN {X -124.831,Y 50.8001,Z 187,A 160.0356,B 2.4036,C 0.0835,E1 2.2573,E2 293.4559} C_DIS
LIN {X -126.094,Y 47.5778,Z 187,A 161.8295,B 2.4036,C 0.0866,E1 2.2554,E2 291.6237} C_DIS
LIN {X -127.2107,Y 44.5066,Z 187,A 163.4209,B 2.4034,C 0.0898,E1 2.2539,E2 290.0086} C_DIS
LIN {X -128.7294,Y 39.9026,Z 187,A 165.4133,B 2.4032,C 0.0954,E1 2.2522,E2 288.0261} C_DIS
LIN {X -129.5984,Y 36.9869,Z 187,A 167.0614,B 2.4031,C 0.0982,E1 2.2509,E2 286.3353} C_DIS
LIN {X -131.0517,Y 31.4442,Z 187,A 170.304,B 2.4029,C 0.1031,E1 2.2487,E2 282.9942} C_DIS
LIN {X -132.3783,Y 25.2839,Z 187,A 172.1055,B 2.4025,C 0.1123,E1 2.2478,E2 281.3036} C_DIS
LIN {X -132.8893,Y 22.4458,Z 187,A 173.3915,B 2.4023,C 0.1156,E1 2.2472,E2 280.011} C_DIS
LIN {X -133.3954,Y 19.2093,Z 187,A 175.0193,B 2.4021,C 0.1189,E1 2.2465,E2 278.3551} C_DIS
LIN {X -133.8825,Y 15.4618,Z 187,A 176.6973,B 2.4019,C 0.1233,E1 2.2459,E2 276.6693} C_DIS
LIN {X -134.2341,Y 12.0432,Z 187,A 178.3946,B 2.4017,C 0.1269,E1 2.2454,E2 274.9437} C_DIS
LIN {X -134.5461,Y 7.8049,Z 187,A -179.7353,B 2.4015,C 0.1318,E1 2.2451,E2 273.0668} C_DIS
LIN {X -134.7162,Y 3.862,Z 187,A -178.0086,B 2.4012,C 0.1364,E1 2.2449,E2 271.335} C_DIS
LIN {X -134.7717,Y 0.3098,Z 187,A -176.2807,B 2.401,C 0.1402,E1 2.2449,E2 269.5808} C_DIS
LIN {X -134.7171,Y -3.8308,Z 187,A -174.5137,B 2.4007,C 0.1451,E1 2.2449,E2 267.814} C_DIS
LIN {X -134.563,Y -7.5306,Z 187,A -172.7187,B 2.4005,C 0.1491,E1 2.2453,E2 265.9923} C_DIS
LIN {X -134.2803,Y -11.4956,Z 187,A -171.0409,B 2.4002,C 0.1538,E1 2.2456,E2 264.317} C_DIS
LIN {X -133.9022,Y -15.296,Z 187,A -169.4205,B 2.3999,C 0.1584,E1 2.2461,E2 262.698} C_DIS
LIN {X -133.4861,Y -18.5748,Z 187,A -167.7698,B 2.3996,C 0.1617,E1 2.2467,E2 261.0171} C_DIS
LIN {X -132.8975,Y -22.3967,Z 187,A -166.0872,B 2.3993,C 0.1662,E1 2.2475,E2 259.3305} C_DIS
LIN {X -132.1674,Y -26.3691,Z 187,A -164.2123,B 2.399,C 0.1706,E1 2.2485,E2 257.4365} C_DIS
LIN {X -131.3876,Y -30.0097,Z 187,A -162.7377,B 2.3987,C 0.1751,E1 2.2493,E2 255.9764} C_DIS
LIN {X -130.6975,Y -32.8864,Z 187,A -161.4361,B 2.3984,C 0.1784,E1 2.2502,E2 254.6698} C_DIS
LIN {X -130.0072,Y -35.5251,Z 187,A -159.8606,B 2.3983,C 0.1806,E1 2.2514,E2 253.0421} C_DIS
LIN {X -128.8649,Y -39.46,Z 187,A -157.5606,B 2.398,C 0.1839,E1 2.2533,E2 250.6713} C_DIS
LIN {X -127.3673,Y -44.0547,Z 187,A -156.194,B 2.3975,C 0.191,E1 2.2545,E2 249.3939} C_DIS
LIN {X -126.4968,Y -46.5023,Z 187,A -154.5998,B 2.3973,C 0.1927,E1 2.2561,E2 247.7375} C_DIS
LIN {X -124.6687,Y -51.2012,Z 187,A -152.4493,B 2.3969,C 0.1981,E1 2.2583,E2 245.587} C_DIS
LIN {X -123.3049,Y -54.402,Z 187,A -150.9068,B 2.3966,C 0.2017,E1 2.26,E2 244.0369} C_DIS
LIN {X -121.8388,Y -57.6091,Z 187,A -149.3555,B 2.3963,C 0.2053,E1 2.2619,E2 242.4794} C_DIS
LIN {X -120.315,Y -60.7267,Z 187,A -148.0248,B 2.3959,C 0.2094,E1 2.2635,E2 241.1678} C_DIS
LIN {X -118.6452,Y -63.9304,Z 187,A -146.1673,B 2.3957,C 0.2122,E1 2.266,E2 239.2696} C_DIS
Enddeposition()
END
